REGION Network 19: 9
   RUNG wire#powerrail
      I_Contact( "AlwaysFALSE" )
      Contact( "DB_Data".F9.Sensor_Correct_Position )
      wire#w1
      Contact( "Q_Door_Open" )
      { S7_Templates := "SrcType := Int" } LT_Contact(in1 := "Simu_Door_F9", in2 := 10)
      Contact( "Clock_1Hz" )
      P_Trig( "P108" )
      Add(in1 := "Simu_Door_F9", in2 := 1, out => "Simu_Door_F9")
   END_RUNG
   RUNG wire#w1
      Contact( "Q_Door_Close" )
      { S7_Templates := "SrcType := Int" } GT_Contact(in1 := "Simu_Door_F9", in2 := 0)
      Contact( "Clock_1Hz" )
      P_Trig( "P109" )
      Sub(in1 := "Simu_Door_F9", in2 := 1, out => "Simu_Door_F9")
   END_RUNG
   // the same network as SCL:
   #_w1 := NOT "AlwaysFALSE" AND "DB_Data".F9.Sensor_Correct_Position;
   #_w2 := #_w1 AND "Q_Door_Open" AND ("Simu_Door_F9" < 10) AND "Clock_1Hz";
   #_w3 := #_w2 AND NOT "P108";   // rising edge
   "P108" := #_w2;
   IF #_w3 THEN "Simu_Door_F9" := "Simu_Door_F9" + 1; END_IF;
   #_w4 := #_w1 AND "Q_Door_Close" AND ("Simu_Door_F9" > 0) AND "Clock_1Hz";
   #_w5 := #_w4 AND NOT "P109";   // rising edge
   "P109" := #_w4;
   IF #_w5 THEN "Simu_Door_F9" := "Simu_Door_F9" - 1; END_IF;
END_REGION

REGION Network 20: 9
   RUNG wire#powerrail
      I_Contact( "AlwaysFALSE" )
      Contact( "DB_Data".F9.Position )
      wire#w1
      { S7_Templates := "SrcType := Int" } GE_Contact(in1 := "Simu_Door_F9", in2 := 10)
      Coil( "DB_Data".F9.Door_Opened )
   END_RUNG
   RUNG wire#w1
      { S7_Templates := "SrcType := Int" } LE_Contact(in1 := "Simu_Door_F9", in2 := 0)
      Coil( "DB_Data".F9.Door_Closed )
   END_RUNG
   // the same network as SCL:
   #_w1 := NOT "AlwaysFALSE" AND "DB_Data".F9.Position;
   "DB_Data".F9.Door_Opened := #_w1 AND ("Simu_Door_F9" >= 10);
   "DB_Data".F9.Door_Closed := #_w1 AND ("Simu_Door_F9" <= 0);
END_REGION

REGION Network 21: 10
   RUNG wire#powerrail
      I_Contact( "AlwaysFALSE" )
      Contact( "DB_Data".F10.Sensor_Correct_Position )
      wire#w1
      Contact( "Q_Door_Open" )
      { S7_Templates := "SrcType := Int" } LT_Contact(in1 := "Simu_Door_F10", in2 := 10)
      Contact( "Clock_1Hz" )
      P_Trig( "P110" )
      Add(in1 := "Simu_Door_F10", in2 := 1, out => "Simu_Door_F10")
   END_RUNG
   RUNG wire#w1
      Contact( "Q_Door_Close" )
      { S7_Templates := "SrcType := Int" } GT_Contact(in1 := "Simu_Door_F10", in2 := 0)
      Contact( "Clock_1Hz" )
      P_Trig( "P111" )
      Sub(in1 := "Simu_Door_F10", in2 := 1, out => "Simu_Door_F10")
   END_RUNG
   // the same network as SCL:
   #_w1 := NOT "AlwaysFALSE" AND "DB_Data".F10.Sensor_Correct_Position;
   #_w2 := #_w1 AND "Q_Door_Open" AND ("Simu_Door_F10" < 10) AND "Clock_1Hz";
   #_w3 := #_w2 AND NOT "P110";   // rising edge
   "P110" := #_w2;
   IF #_w3 THEN "Simu_Door_F10" := "Simu_Door_F10" + 1; END_IF;
   #_w4 := #_w1 AND "Q_Door_Close" AND ("Simu_Door_F10" > 0) AND "Clock_1Hz";
   #_w5 := #_w4 AND NOT "P111";   // rising edge
   "P111" := #_w4;
   IF #_w5 THEN "Simu_Door_F10" := "Simu_Door_F10" - 1; END_IF;
END_REGION

REGION Network 22: 10
   RUNG wire#powerrail
      I_Contact( "AlwaysFALSE" )
      Contact( "DB_Data".F10.Position )
      wire#w1
      { S7_Templates := "SrcType := Int" } GE_Contact(in1 := "Simu_Door_F10", in2 := 10)
      Coil( "DB_Data".F10.Door_Opened )
   END_RUNG
   RUNG wire#w1
      { S7_Templates := "SrcType := Int" } LE_Contact(in1 := "Simu_Door_F10", in2 := 0)
      Coil( "DB_Data".F10.Door_Closed )
   END_RUNG
   // the same network as SCL:
   #_w1 := NOT "AlwaysFALSE" AND "DB_Data".F10.Position;
   "DB_Data".F10.Door_Opened := #_w1 AND ("Simu_Door_F10" >= 10);
   "DB_Data".F10.Door_Closed := #_w1 AND ("Simu_Door_F10" <= 0);
END_REGION

REGION Network 23: 11
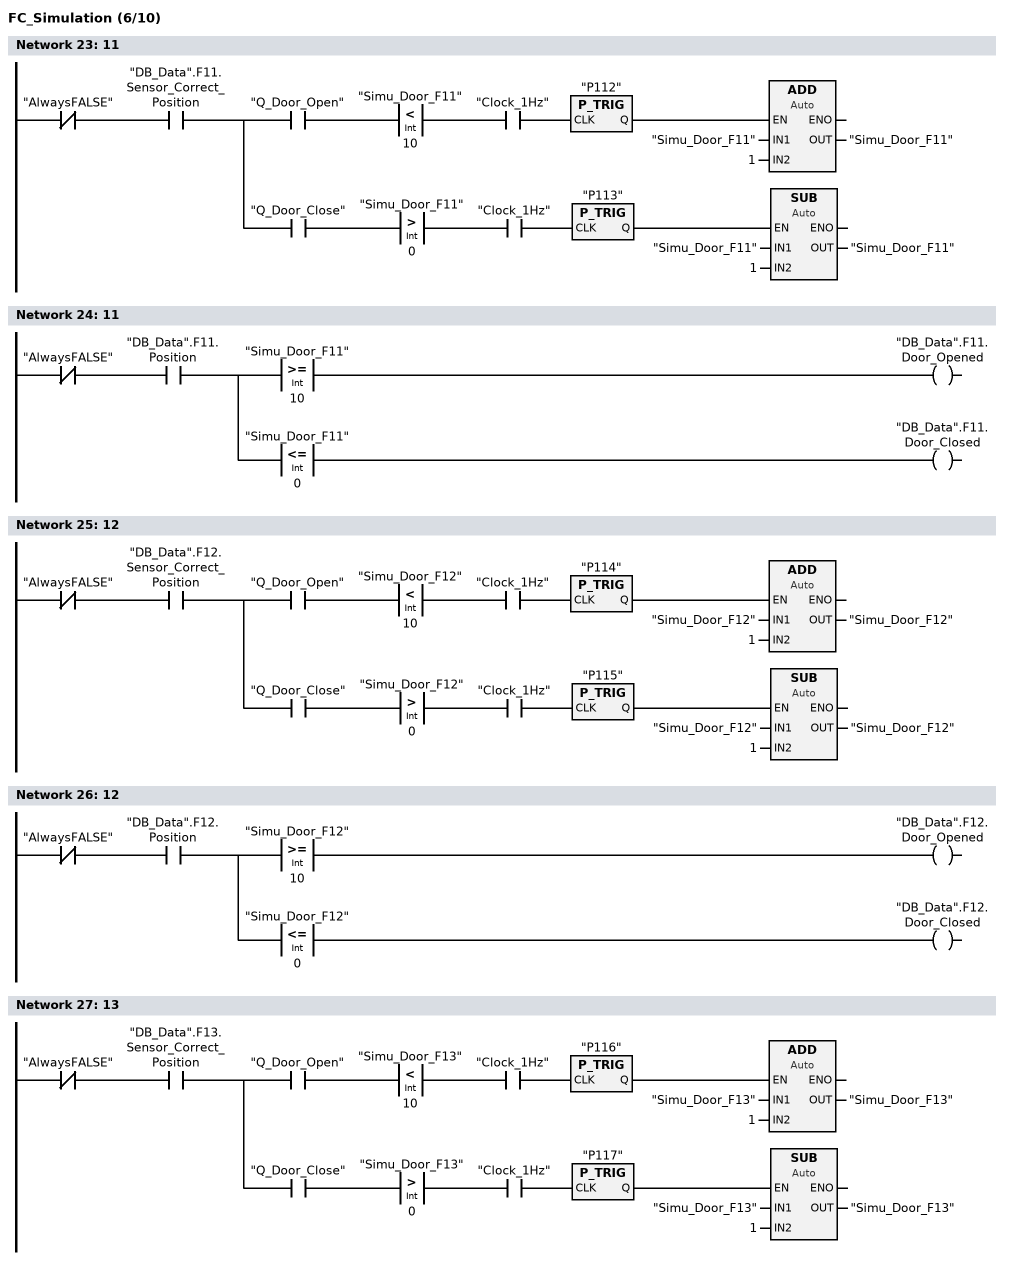
   RUNG wire#powerrail
      I_Contact( "AlwaysFALSE" )
      Contact( "DB_Data".F11.Sensor_Correct_Position )
      wire#w1
      Contact( "Q_Door_Open" )
      { S7_Templates := "SrcType := Int" } LT_Contact(in1 := "Simu_Door_F11", in2 := 10)
      Contact( "Clock_1Hz" )
      P_Trig( "P112" )
      Add(in1 := "Simu_Door_F11", in2 := 1, out => "Simu_Door_F11")
   END_RUNG
   RUNG wire#w1
      Contact( "Q_Door_Close" )
      { S7_Templates := "SrcType := Int" } GT_Contact(in1 := "Simu_Door_F11", in2 := 0)
      Contact( "Clock_1Hz" )
      P_Trig( "P113" )
      Sub(in1 := "Simu_Door_F11", in2 := 1, out => "Simu_Door_F11")
   END_RUNG
   // the same network as SCL:
   #_w1 := NOT "AlwaysFALSE" AND "DB_Data".F11.Sensor_Correct_Position;
   #_w2 := #_w1 AND "Q_Door_Open" AND ("Simu_Door_F11" < 10) AND "Clock_1Hz";
   #_w3 := #_w2 AND NOT "P112";   // rising edge
   "P112" := #_w2;
   IF #_w3 THEN "Simu_Door_F11" := "Simu_Door_F11" + 1; END_IF;
   #_w4 := #_w1 AND "Q_Door_Close" AND ("Simu_Door_F11" > 0) AND "Clock_1Hz";
   #_w5 := #_w4 AND NOT "P113";   // rising edge
   "P113" := #_w4;
   IF #_w5 THEN "Simu_Door_F11" := "Simu_Door_F11" - 1; END_IF;
END_REGION

REGION Network 24: 11
   RUNG wire#powerrail
      I_Contact( "AlwaysFALSE" )
      Contact( "DB_Data".F11.Position )
      wire#w1
      { S7_Templates := "SrcType := Int" } GE_Contact(in1 := "Simu_Door_F11", in2 := 10)
      Coil( "DB_Data".F11.Door_Opened )
   END_RUNG
   RUNG wire#w1
      { S7_Templates := "SrcType := Int" } LE_Contact(in1 := "Simu_Door_F11", in2 := 0)
      Coil( "DB_Data".F11.Door_Closed )
   END_RUNG
   // the same network as SCL:
   #_w1 := NOT "AlwaysFALSE" AND "DB_Data".F11.Position;
   "DB_Data".F11.Door_Opened := #_w1 AND ("Simu_Door_F11" >= 10);
   "DB_Data".F11.Door_Closed := #_w1 AND ("Simu_Door_F11" <= 0);
END_REGION

REGION Network 25: 12
   RUNG wire#powerrail
      I_Contact( "AlwaysFALSE" )
      Contact( "DB_Data".F12.Sensor_Correct_Position )
      wire#w1
      Contact( "Q_Door_Open" )
      { S7_Templates := "SrcType := Int" } LT_Contact(in1 := "Simu_Door_F12", in2 := 10)
      Contact( "Clock_1Hz" )
      P_Trig( "P114" )
      Add(in1 := "Simu_Door_F12", in2 := 1, out => "Simu_Door_F12")
   END_RUNG
   RUNG wire#w1
      Contact( "Q_Door_Close" )
      { S7_Templates := "SrcType := Int" } GT_Contact(in1 := "Simu_Door_F12", in2 := 0)
      Contact( "Clock_1Hz" )
      P_Trig( "P115" )
      Sub(in1 := "Simu_Door_F12", in2 := 1, out => "Simu_Door_F12")
   END_RUNG
   // the same network as SCL:
   #_w1 := NOT "AlwaysFALSE" AND "DB_Data".F12.Sensor_Correct_Position;
   #_w2 := #_w1 AND "Q_Door_Open" AND ("Simu_Door_F12" < 10) AND "Clock_1Hz";
   #_w3 := #_w2 AND NOT "P114";   // rising edge
   "P114" := #_w2;
   IF #_w3 THEN "Simu_Door_F12" := "Simu_Door_F12" + 1; END_IF;
   #_w4 := #_w1 AND "Q_Door_Close" AND ("Simu_Door_F12" > 0) AND "Clock_1Hz";
   #_w5 := #_w4 AND NOT "P115";   // rising edge
   "P115" := #_w4;
   IF #_w5 THEN "Simu_Door_F12" := "Simu_Door_F12" - 1; END_IF;
END_REGION

REGION Network 26: 12
   RUNG wire#powerrail
      I_Contact( "AlwaysFALSE" )
      Contact( "DB_Data".F12.Position )
      wire#w1
      { S7_Templates := "SrcType := Int" } GE_Contact(in1 := "Simu_Door_F12", in2 := 10)
      Coil( "DB_Data".F12.Door_Opened )
   END_RUNG
   RUNG wire#w1
      { S7_Templates := "SrcType := Int" } LE_Contact(in1 := "Simu_Door_F12", in2 := 0)
      Coil( "DB_Data".F12.Door_Closed )
   END_RUNG
   // the same network as SCL:
   #_w1 := NOT "AlwaysFALSE" AND "DB_Data".F12.Position;
   "DB_Data".F12.Door_Opened := #_w1 AND ("Simu_Door_F12" >= 10);
   "DB_Data".F12.Door_Closed := #_w1 AND ("Simu_Door_F12" <= 0);
END_REGION

REGION Network 27: 13
   RUNG wire#powerrail
      I_Contact( "AlwaysFALSE" )
      Contact( "DB_Data".F13.Sensor_Correct_Position )
      wire#w1
      Contact( "Q_Door_Open" )
      { S7_Templates := "SrcType := Int" } LT_Contact(in1 := "Simu_Door_F13", in2 := 10)
      Contact( "Clock_1Hz" )
      P_Trig( "P116" )
      Add(in1 := "Simu_Door_F13", in2 := 1, out => "Simu_Door_F13")
   END_RUNG
   RUNG wire#w1
      Contact( "Q_Door_Close" )
      { S7_Templates := "SrcType := Int" } GT_Contact(in1 := "Simu_Door_F13", in2 := 0)
      Contact( "Clock_1Hz" )
      P_Trig( "P117" )
      Sub(in1 := "Simu_Door_F13", in2 := 1, out => "Simu_Door_F13")
   END_RUNG
   // the same network as SCL:
   #_w1 := NOT "AlwaysFALSE" AND "DB_Data".F13.Sensor_Correct_Position;
   #_w2 := #_w1 AND "Q_Door_Open" AND ("Simu_Door_F13" < 10) AND "Clock_1Hz";
   #_w3 := #_w2 AND NOT "P116";   // rising edge
   "P116" := #_w2;
   IF #_w3 THEN "Simu_Door_F13" := "Simu_Door_F13" + 1; END_IF;
   #_w4 := #_w1 AND "Q_Door_Close" AND ("Simu_Door_F13" > 0) AND "Clock_1Hz";
   #_w5 := #_w4 AND NOT "P117";   // rising edge
   "P117" := #_w4;
   IF #_w5 THEN "Simu_Door_F13" := "Simu_Door_F13" - 1; END_IF;
END_REGION

REGION Network 28: 13
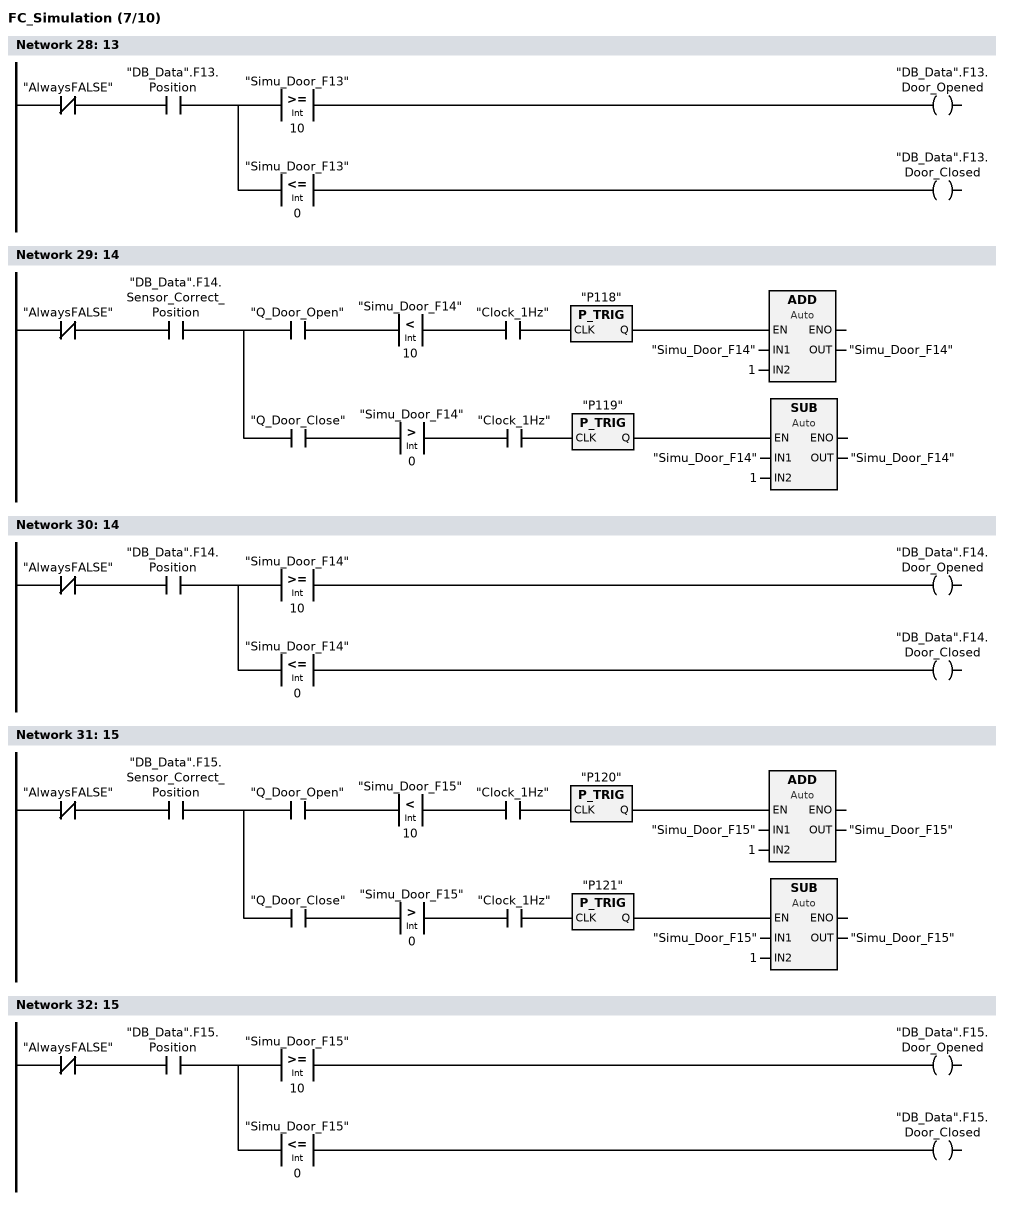
   RUNG wire#powerrail
      I_Contact( "AlwaysFALSE" )
      Contact( "DB_Data".F13.Position )
      wire#w1
      { S7_Templates := "SrcType := Int" } GE_Contact(in1 := "Simu_Door_F13", in2 := 10)
      Coil( "DB_Data".F13.Door_Opened )
   END_RUNG
   RUNG wire#w1
      { S7_Templates := "SrcType := Int" } LE_Contact(in1 := "Simu_Door_F13", in2 := 0)
      Coil( "DB_Data".F13.Door_Closed )
   END_RUNG
   // the same network as SCL:
   #_w1 := NOT "AlwaysFALSE" AND "DB_Data".F13.Position;
   "DB_Data".F13.Door_Opened := #_w1 AND ("Simu_Door_F13" >= 10);
   "DB_Data".F13.Door_Closed := #_w1 AND ("Simu_Door_F13" <= 0);
END_REGION

REGION Network 29: 14
   RUNG wire#powerrail
      I_Contact( "AlwaysFALSE" )
      Contact( "DB_Data".F14.Sensor_Correct_Position )
      wire#w1
      Contact( "Q_Door_Open" )
      { S7_Templates := "SrcType := Int" } LT_Contact(in1 := "Simu_Door_F14", in2 := 10)
      Contact( "Clock_1Hz" )
      P_Trig( "P118" )
      Add(in1 := "Simu_Door_F14", in2 := 1, out => "Simu_Door_F14")
   END_RUNG
   RUNG wire#w1
      Contact( "Q_Door_Close" )
      { S7_Templates := "SrcType := Int" } GT_Contact(in1 := "Simu_Door_F14", in2 := 0)
      Contact( "Clock_1Hz" )
      P_Trig( "P119" )
      Sub(in1 := "Simu_Door_F14", in2 := 1, out => "Simu_Door_F14")
   END_RUNG
   // the same network as SCL:
   #_w1 := NOT "AlwaysFALSE" AND "DB_Data".F14.Sensor_Correct_Position;
   #_w2 := #_w1 AND "Q_Door_Open" AND ("Simu_Door_F14" < 10) AND "Clock_1Hz";
   #_w3 := #_w2 AND NOT "P118";   // rising edge
   "P118" := #_w2;
   IF #_w3 THEN "Simu_Door_F14" := "Simu_Door_F14" + 1; END_IF;
   #_w4 := #_w1 AND "Q_Door_Close" AND ("Simu_Door_F14" > 0) AND "Clock_1Hz";
   #_w5 := #_w4 AND NOT "P119";   // rising edge
   "P119" := #_w4;
   IF #_w5 THEN "Simu_Door_F14" := "Simu_Door_F14" - 1; END_IF;
END_REGION

REGION Network 30: 14
   RUNG wire#powerrail
      I_Contact( "AlwaysFALSE" )
      Contact( "DB_Data".F14.Position )
      wire#w1
      { S7_Templates := "SrcType := Int" } GE_Contact(in1 := "Simu_Door_F14", in2 := 10)
      Coil( "DB_Data".F14.Door_Opened )
   END_RUNG
   RUNG wire#w1
      { S7_Templates := "SrcType := Int" } LE_Contact(in1 := "Simu_Door_F14", in2 := 0)
      Coil( "DB_Data".F14.Door_Closed )
   END_RUNG
   // the same network as SCL:
   #_w1 := NOT "AlwaysFALSE" AND "DB_Data".F14.Position;
   "DB_Data".F14.Door_Opened := #_w1 AND ("Simu_Door_F14" >= 10);
   "DB_Data".F14.Door_Closed := #_w1 AND ("Simu_Door_F14" <= 0);
END_REGION

REGION Network 31: 15
   RUNG wire#powerrail
      I_Contact( "AlwaysFALSE" )
      Contact( "DB_Data".F15.Sensor_Correct_Position )
      wire#w1
      Contact( "Q_Door_Open" )
      { S7_Templates := "SrcType := Int" } LT_Contact(in1 := "Simu_Door_F15", in2 := 10)
      Contact( "Clock_1Hz" )
      P_Trig( "P120" )
      Add(in1 := "Simu_Door_F15", in2 := 1, out => "Simu_Door_F15")
   END_RUNG
   RUNG wire#w1
      Contact( "Q_Door_Close" )
      { S7_Templates := "SrcType := Int" } GT_Contact(in1 := "Simu_Door_F15", in2 := 0)
      Contact( "Clock_1Hz" )
      P_Trig( "P121" )
      Sub(in1 := "Simu_Door_F15", in2 := 1, out => "Simu_Door_F15")
   END_RUNG
   // the same network as SCL:
   #_w1 := NOT "AlwaysFALSE" AND "DB_Data".F15.Sensor_Correct_Position;
   #_w2 := #_w1 AND "Q_Door_Open" AND ("Simu_Door_F15" < 10) AND "Clock_1Hz";
   #_w3 := #_w2 AND NOT "P120";   // rising edge
   "P120" := #_w2;
   IF #_w3 THEN "Simu_Door_F15" := "Simu_Door_F15" + 1; END_IF;
   #_w4 := #_w1 AND "Q_Door_Close" AND ("Simu_Door_F15" > 0) AND "Clock_1Hz";
   #_w5 := #_w4 AND NOT "P121";   // rising edge
   "P121" := #_w4;
   IF #_w5 THEN "Simu_Door_F15" := "Simu_Door_F15" - 1; END_IF;
END_REGION

REGION Network 32: 15
   RUNG wire#powerrail
      I_Contact( "AlwaysFALSE" )
      Contact( "DB_Data".F15.Position )
      wire#w1
      { S7_Templates := "SrcType := Int" } GE_Contact(in1 := "Simu_Door_F15", in2 := 10)
      Coil( "DB_Data".F15.Door_Opened )
   END_RUNG
   RUNG wire#w1
      { S7_Templates := "SrcType := Int" } LE_Contact(in1 := "Simu_Door_F15", in2 := 0)
      Coil( "DB_Data".F15.Door_Closed )
   END_RUNG
   // the same network as SCL:
   #_w1 := NOT "AlwaysFALSE" AND "DB_Data".F15.Position;
   "DB_Data".F15.Door_Opened := #_w1 AND ("Simu_Door_F15" >= 10);
   "DB_Data".F15.Door_Closed := #_w1 AND ("Simu_Door_F15" <= 0);
END_REGION

REGION Network 33: 16
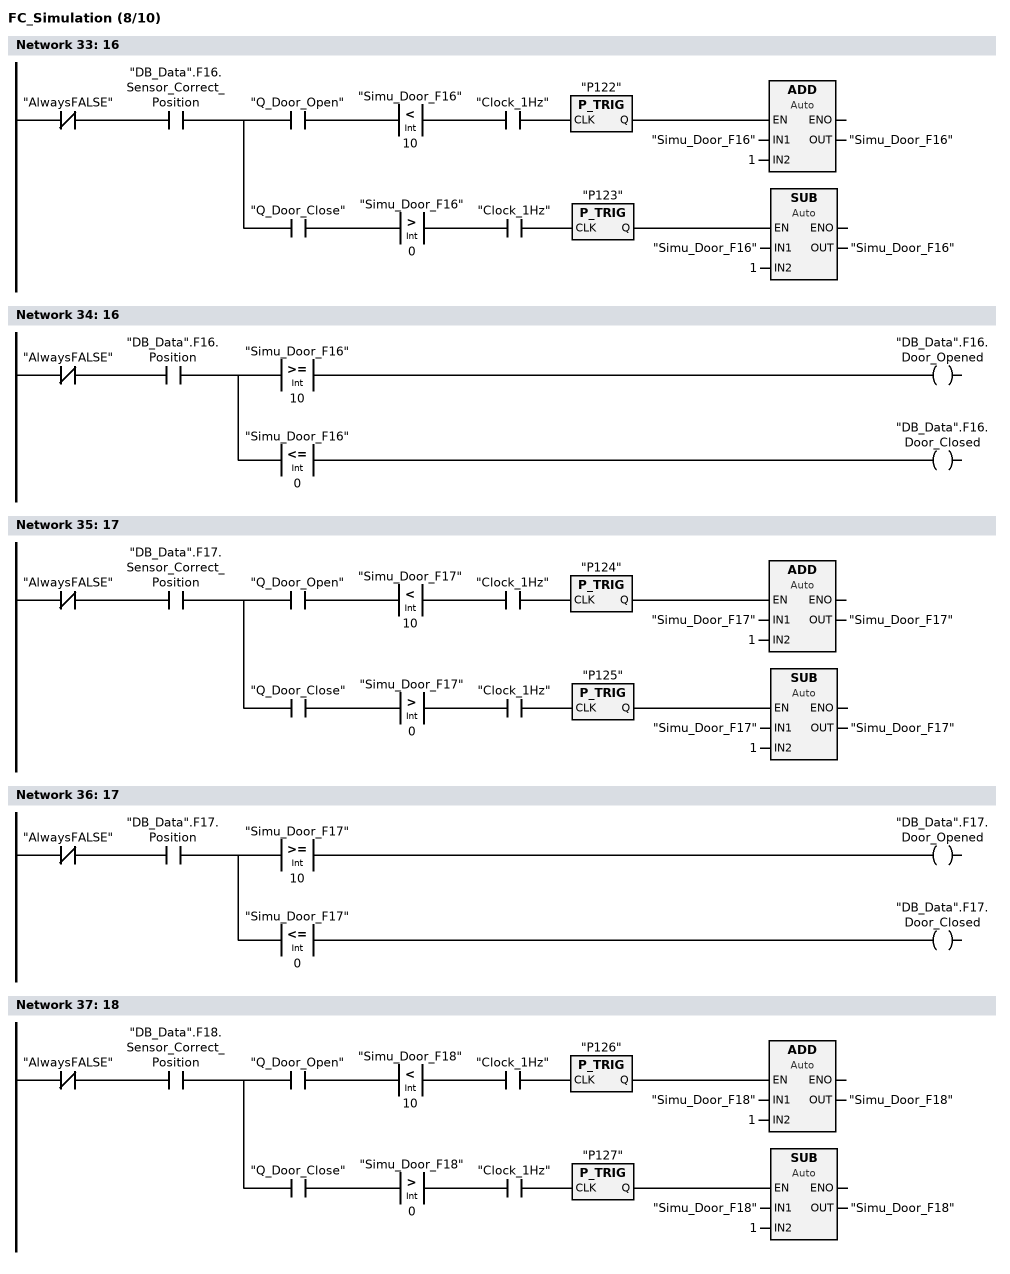
   RUNG wire#powerrail
      I_Contact( "AlwaysFALSE" )
      Contact( "DB_Data".F16.Sensor_Correct_Position )
      wire#w1
      Contact( "Q_Door_Open" )
      { S7_Templates := "SrcType := Int" } LT_Contact(in1 := "Simu_Door_F16", in2 := 10)
      Contact( "Clock_1Hz" )
      P_Trig( "P122" )
      Add(in1 := "Simu_Door_F16", in2 := 1, out => "Simu_Door_F16")
   END_RUNG
   RUNG wire#w1
      Contact( "Q_Door_Close" )
      { S7_Templates := "SrcType := Int" } GT_Contact(in1 := "Simu_Door_F16", in2 := 0)
      Contact( "Clock_1Hz" )
      P_Trig( "P123" )
      Sub(in1 := "Simu_Door_F16", in2 := 1, out => "Simu_Door_F16")
   END_RUNG
   // the same network as SCL:
   #_w1 := NOT "AlwaysFALSE" AND "DB_Data".F16.Sensor_Correct_Position;
   #_w2 := #_w1 AND "Q_Door_Open" AND ("Simu_Door_F16" < 10) AND "Clock_1Hz";
   #_w3 := #_w2 AND NOT "P122";   // rising edge
   "P122" := #_w2;
   IF #_w3 THEN "Simu_Door_F16" := "Simu_Door_F16" + 1; END_IF;
   #_w4 := #_w1 AND "Q_Door_Close" AND ("Simu_Door_F16" > 0) AND "Clock_1Hz";
   #_w5 := #_w4 AND NOT "P123";   // rising edge
   "P123" := #_w4;
   IF #_w5 THEN "Simu_Door_F16" := "Simu_Door_F16" - 1; END_IF;
END_REGION

REGION Network 34: 16
   RUNG wire#powerrail
      I_Contact( "AlwaysFALSE" )
      Contact( "DB_Data".F16.Position )
      wire#w1
      { S7_Templates := "SrcType := Int" } GE_Contact(in1 := "Simu_Door_F16", in2 := 10)
      Coil( "DB_Data".F16.Door_Opened )
   END_RUNG
   RUNG wire#w1
      { S7_Templates := "SrcType := Int" } LE_Contact(in1 := "Simu_Door_F16", in2 := 0)
      Coil( "DB_Data".F16.Door_Closed )
   END_RUNG
   // the same network as SCL:
   #_w1 := NOT "AlwaysFALSE" AND "DB_Data".F16.Position;
   "DB_Data".F16.Door_Opened := #_w1 AND ("Simu_Door_F16" >= 10);
   "DB_Data".F16.Door_Closed := #_w1 AND ("Simu_Door_F16" <= 0);
END_REGION

REGION Network 35: 17
   RUNG wire#powerrail
      I_Contact( "AlwaysFALSE" )
      Contact( "DB_Data".F17.Sensor_Correct_Position )
      wire#w1
      Contact( "Q_Door_Open" )
      { S7_Templates := "SrcType := Int" } LT_Contact(in1 := "Simu_Door_F17", in2 := 10)
      Contact( "Clock_1Hz" )
      P_Trig( "P124" )
      Add(in1 := "Simu_Door_F17", in2 := 1, out => "Simu_Door_F17")
   END_RUNG
   RUNG wire#w1
      Contact( "Q_Door_Close" )
      { S7_Templates := "SrcType := Int" } GT_Contact(in1 := "Simu_Door_F17", in2 := 0)
      Contact( "Clock_1Hz" )
      P_Trig( "P125" )
      Sub(in1 := "Simu_Door_F17", in2 := 1, out => "Simu_Door_F17")
   END_RUNG
   // the same network as SCL:
   #_w1 := NOT "AlwaysFALSE" AND "DB_Data".F17.Sensor_Correct_Position;
   #_w2 := #_w1 AND "Q_Door_Open" AND ("Simu_Door_F17" < 10) AND "Clock_1Hz";
   #_w3 := #_w2 AND NOT "P124";   // rising edge
   "P124" := #_w2;
   IF #_w3 THEN "Simu_Door_F17" := "Simu_Door_F17" + 1; END_IF;
   #_w4 := #_w1 AND "Q_Door_Close" AND ("Simu_Door_F17" > 0) AND "Clock_1Hz";
   #_w5 := #_w4 AND NOT "P125";   // rising edge
   "P125" := #_w4;
   IF #_w5 THEN "Simu_Door_F17" := "Simu_Door_F17" - 1; END_IF;
END_REGION

REGION Network 36: 17
   RUNG wire#powerrail
      I_Contact( "AlwaysFALSE" )
      Contact( "DB_Data".F17.Position )
      wire#w1
      { S7_Templates := "SrcType := Int" } GE_Contact(in1 := "Simu_Door_F17", in2 := 10)
      Coil( "DB_Data".F17.Door_Opened )
   END_RUNG
   RUNG wire#w1
      { S7_Templates := "SrcType := Int" } LE_Contact(in1 := "Simu_Door_F17", in2 := 0)
      Coil( "DB_Data".F17.Door_Closed )
   END_RUNG
   // the same network as SCL:
   #_w1 := NOT "AlwaysFALSE" AND "DB_Data".F17.Position;
   "DB_Data".F17.Door_Opened := #_w1 AND ("Simu_Door_F17" >= 10);
   "DB_Data".F17.Door_Closed := #_w1 AND ("Simu_Door_F17" <= 0);
END_REGION

REGION Network 37: 18
   RUNG wire#powerrail
      I_Contact( "AlwaysFALSE" )
      Contact( "DB_Data".F18.Sensor_Correct_Position )
      wire#w1
      Contact( "Q_Door_Open" )
      { S7_Templates := "SrcType := Int" } LT_Contact(in1 := "Simu_Door_F18", in2 := 10)
      Contact( "Clock_1Hz" )
      P_Trig( "P126" )
      Add(in1 := "Simu_Door_F18", in2 := 1, out => "Simu_Door_F18")
   END_RUNG
   RUNG wire#w1
      Contact( "Q_Door_Close" )
      { S7_Templates := "SrcType := Int" } GT_Contact(in1 := "Simu_Door_F18", in2 := 0)
      Contact( "Clock_1Hz" )
      P_Trig( "P127" )
      Sub(in1 := "Simu_Door_F18", in2 := 1, out => "Simu_Door_F18")
   END_RUNG
   // the same network as SCL:
   #_w1 := NOT "AlwaysFALSE" AND "DB_Data".F18.Sensor_Correct_Position;
   #_w2 := #_w1 AND "Q_Door_Open" AND ("Simu_Door_F18" < 10) AND "Clock_1Hz";
   #_w3 := #_w2 AND NOT "P126";   // rising edge
   "P126" := #_w2;
   IF #_w3 THEN "Simu_Door_F18" := "Simu_Door_F18" + 1; END_IF;
   #_w4 := #_w1 AND "Q_Door_Close" AND ("Simu_Door_F18" > 0) AND "Clock_1Hz";
   #_w5 := #_w4 AND NOT "P127";   // rising edge
   "P127" := #_w4;
   IF #_w5 THEN "Simu_Door_F18" := "Simu_Door_F18" - 1; END_IF;
END_REGION

REGION Network 38: 18
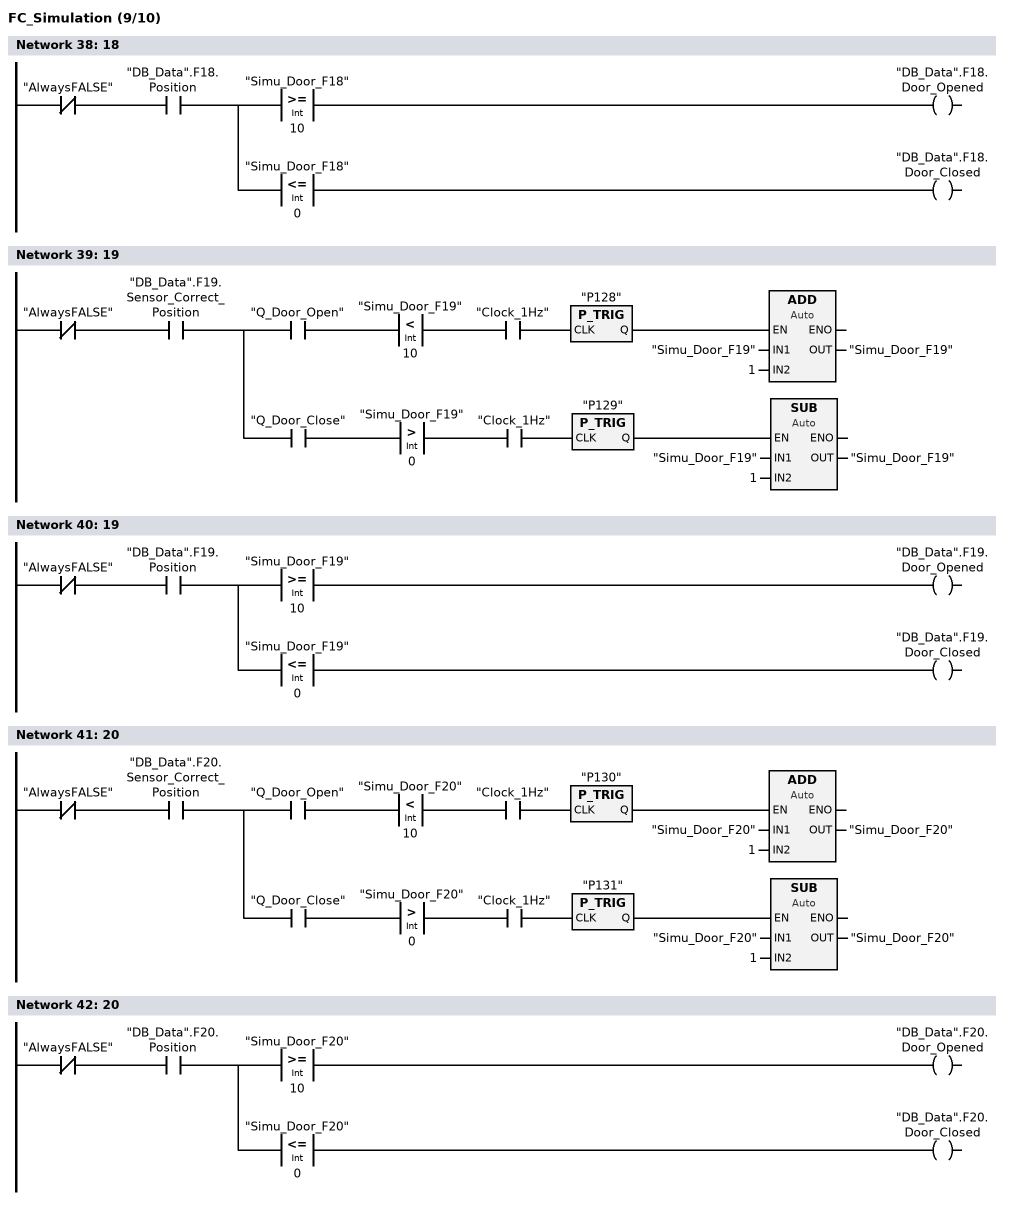
   RUNG wire#powerrail
      I_Contact( "AlwaysFALSE" )
      Contact( "DB_Data".F18.Position )
      wire#w1
      { S7_Templates := "SrcType := Int" } GE_Contact(in1 := "Simu_Door_F18", in2 := 10)
      Coil( "DB_Data".F18.Door_Opened )
   END_RUNG
   RUNG wire#w1
      { S7_Templates := "SrcType := Int" } LE_Contact(in1 := "Simu_Door_F18", in2 := 0)
      Coil( "DB_Data".F18.Door_Closed )
   END_RUNG
   // the same network as SCL:
   #_w1 := NOT "AlwaysFALSE" AND "DB_Data".F18.Position;
   "DB_Data".F18.Door_Opened := #_w1 AND ("Simu_Door_F18" >= 10);
   "DB_Data".F18.Door_Closed := #_w1 AND ("Simu_Door_F18" <= 0);
END_REGION

REGION Network 39: 19
   RUNG wire#powerrail
      I_Contact( "AlwaysFALSE" )
      Contact( "DB_Data".F19.Sensor_Correct_Position )
      wire#w1
      Contact( "Q_Door_Open" )
      { S7_Templates := "SrcType := Int" } LT_Contact(in1 := "Simu_Door_F19", in2 := 10)
      Contact( "Clock_1Hz" )
      P_Trig( "P128" )
      Add(in1 := "Simu_Door_F19", in2 := 1, out => "Simu_Door_F19")
   END_RUNG
   RUNG wire#w1
      Contact( "Q_Door_Close" )
      { S7_Templates := "SrcType := Int" } GT_Contact(in1 := "Simu_Door_F19", in2 := 0)
      Contact( "Clock_1Hz" )
      P_Trig( "P129" )
      Sub(in1 := "Simu_Door_F19", in2 := 1, out => "Simu_Door_F19")
   END_RUNG
   // the same network as SCL:
   #_w1 := NOT "AlwaysFALSE" AND "DB_Data".F19.Sensor_Correct_Position;
   #_w2 := #_w1 AND "Q_Door_Open" AND ("Simu_Door_F19" < 10) AND "Clock_1Hz";
   #_w3 := #_w2 AND NOT "P128";   // rising edge
   "P128" := #_w2;
   IF #_w3 THEN "Simu_Door_F19" := "Simu_Door_F19" + 1; END_IF;
   #_w4 := #_w1 AND "Q_Door_Close" AND ("Simu_Door_F19" > 0) AND "Clock_1Hz";
   #_w5 := #_w4 AND NOT "P129";   // rising edge
   "P129" := #_w4;
   IF #_w5 THEN "Simu_Door_F19" := "Simu_Door_F19" - 1; END_IF;
END_REGION

REGION Network 40: 19
   RUNG wire#powerrail
      I_Contact( "AlwaysFALSE" )
      Contact( "DB_Data".F19.Position )
      wire#w1
      { S7_Templates := "SrcType := Int" } GE_Contact(in1 := "Simu_Door_F19", in2 := 10)
      Coil( "DB_Data".F19.Door_Opened )
   END_RUNG
   RUNG wire#w1
      { S7_Templates := "SrcType := Int" } LE_Contact(in1 := "Simu_Door_F19", in2 := 0)
      Coil( "DB_Data".F19.Door_Closed )
   END_RUNG
   // the same network as SCL:
   #_w1 := NOT "AlwaysFALSE" AND "DB_Data".F19.Position;
   "DB_Data".F19.Door_Opened := #_w1 AND ("Simu_Door_F19" >= 10);
   "DB_Data".F19.Door_Closed := #_w1 AND ("Simu_Door_F19" <= 0);
END_REGION

REGION Network 41: 20
   RUNG wire#powerrail
      I_Contact( "AlwaysFALSE" )
      Contact( "DB_Data".F20.Sensor_Correct_Position )
      wire#w1
      Contact( "Q_Door_Open" )
      { S7_Templates := "SrcType := Int" } LT_Contact(in1 := "Simu_Door_F20", in2 := 10)
      Contact( "Clock_1Hz" )
      P_Trig( "P130" )
      Add(in1 := "Simu_Door_F20", in2 := 1, out => "Simu_Door_F20")
   END_RUNG
   RUNG wire#w1
      Contact( "Q_Door_Close" )
      { S7_Templates := "SrcType := Int" } GT_Contact(in1 := "Simu_Door_F20", in2 := 0)
      Contact( "Clock_1Hz" )
      P_Trig( "P131" )
      Sub(in1 := "Simu_Door_F20", in2 := 1, out => "Simu_Door_F20")
   END_RUNG
   // the same network as SCL:
   #_w1 := NOT "AlwaysFALSE" AND "DB_Data".F20.Sensor_Correct_Position;
   #_w2 := #_w1 AND "Q_Door_Open" AND ("Simu_Door_F20" < 10) AND "Clock_1Hz";
   #_w3 := #_w2 AND NOT "P130";   // rising edge
   "P130" := #_w2;
   IF #_w3 THEN "Simu_Door_F20" := "Simu_Door_F20" + 1; END_IF;
   #_w4 := #_w1 AND "Q_Door_Close" AND ("Simu_Door_F20" > 0) AND "Clock_1Hz";
   #_w5 := #_w4 AND NOT "P131";   // rising edge
   "P131" := #_w4;
   IF #_w5 THEN "Simu_Door_F20" := "Simu_Door_F20" - 1; END_IF;
END_REGION

REGION Network 42: 20
   RUNG wire#powerrail
      I_Contact( "AlwaysFALSE" )
      Contact( "DB_Data".F20.Position )
      wire#w1
      { S7_Templates := "SrcType := Int" } GE_Contact(in1 := "Simu_Door_F20", in2 := 10)
      Coil( "DB_Data".F20.Door_Opened )
   END_RUNG
   RUNG wire#w1
      { S7_Templates := "SrcType := Int" } LE_Contact(in1 := "Simu_Door_F20", in2 := 0)
      Coil( "DB_Data".F20.Door_Closed )
   END_RUNG
   // the same network as SCL:
   #_w1 := NOT "AlwaysFALSE" AND "DB_Data".F20.Position;
   "DB_Data".F20.Door_Opened := #_w1 AND ("Simu_Door_F20" >= 10);
   "DB_Data".F20.Door_Closed := #_w1 AND ("Simu_Door_F20" <= 0);
END_REGION

REGION Network 43: Mô phỏng LS cửa buồng thang
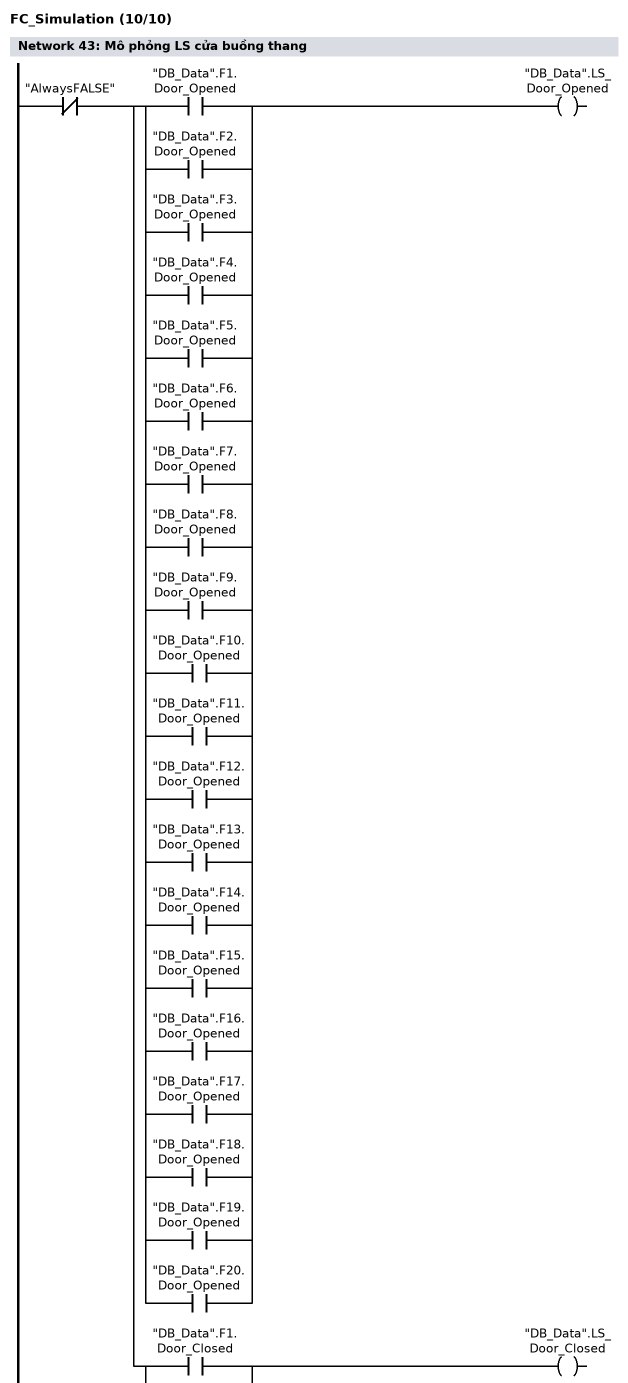
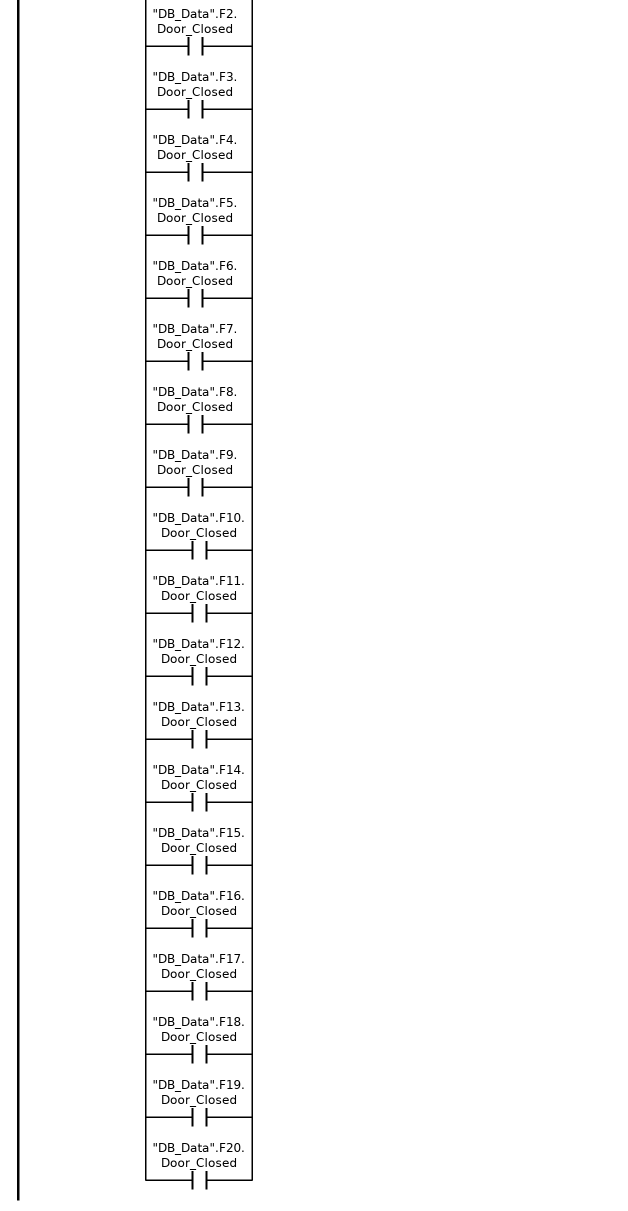
   RUNG wire#powerrail
      I_Contact( "AlwaysFALSE" )
      wire#w1
      Contact( "DB_Data".F1.Door_Opened )
      wire#w2
      Coil( "DB_Data".LS_Door_Opened )
   END_RUNG
   RUNG wire#w1
      Contact( "DB_Data".F2.Door_Opened )
   END_RUNG wire#w2
   RUNG wire#w1
      Contact( "DB_Data".F3.Door_Opened )
   END_RUNG wire#w2
   RUNG wire#w1
      Contact( "DB_Data".F4.Door_Opened )
   END_RUNG wire#w2
   RUNG wire#w1
      Contact( "DB_Data".F5.Door_Opened )
   END_RUNG wire#w2
   RUNG wire#w1
      Contact( "DB_Data".F6.Door_Opened )
   END_RUNG wire#w2
   RUNG wire#w1
      Contact( "DB_Data".F7.Door_Opened )
   END_RUNG wire#w2
   RUNG wire#w1
      Contact( "DB_Data".F8.Door_Opened )
   END_RUNG wire#w2
   RUNG wire#w1
      Contact( "DB_Data".F9.Door_Opened )
   END_RUNG wire#w2
   RUNG wire#w1
      Contact( "DB_Data".F10.Door_Opened )
   END_RUNG wire#w2
   RUNG wire#w1
      Contact( "DB_Data".F11.Door_Opened )
   END_RUNG wire#w2
   RUNG wire#w1
      Contact( "DB_Data".F12.Door_Opened )
   END_RUNG wire#w2
   RUNG wire#w1
      Contact( "DB_Data".F13.Door_Opened )
   END_RUNG wire#w2
   RUNG wire#w1
      Contact( "DB_Data".F14.Door_Opened )
   END_RUNG wire#w2
   RUNG wire#w1
      Contact( "DB_Data".F15.Door_Opened )
   END_RUNG wire#w2
   RUNG wire#w1
      Contact( "DB_Data".F16.Door_Opened )
   END_RUNG wire#w2
   RUNG wire#w1
      Contact( "DB_Data".F17.Door_Opened )
   END_RUNG wire#w2
   RUNG wire#w1
      Contact( "DB_Data".F18.Door_Opened )
   END_RUNG wire#w2
   RUNG wire#w1
      Contact( "DB_Data".F19.Door_Opened )
   END_RUNG wire#w2
   RUNG wire#w1
      Contact( "DB_Data".F20.Door_Opened )
   END_RUNG wire#w2
   RUNG wire#w1
      Contact( "DB_Data".F1.Door_Closed )
      wire#w3
      Coil( "DB_Data".LS_Door_Closed )
   END_RUNG
   RUNG wire#w1
      Contact( "DB_Data".F2.Door_Closed )
   END_RUNG wire#w3
   RUNG wire#w1
      Contact( "DB_Data".F3.Door_Closed )
   END_RUNG wire#w3
   RUNG wire#w1
      Contact( "DB_Data".F4.Door_Closed )
   END_RUNG wire#w3
   RUNG wire#w1
      Contact( "DB_Data".F5.Door_Closed )
   END_RUNG wire#w3
   RUNG wire#w1
      Contact( "DB_Data".F6.Door_Closed )
   END_RUNG wire#w3
   RUNG wire#w1
      Contact( "DB_Data".F7.Door_Closed )
   END_RUNG wire#w3
   RUNG wire#w1
      Contact( "DB_Data".F8.Door_Closed )
   END_RUNG wire#w3
   RUNG wire#w1
      Contact( "DB_Data".F9.Door_Closed )
   END_RUNG wire#w3
   RUNG wire#w1
      Contact( "DB_Data".F10.Door_Closed )
   END_RUNG wire#w3
   RUNG wire#w1
      Contact( "DB_Data".F11.Door_Closed )
   END_RUNG wire#w3
   RUNG wire#w1
      Contact( "DB_Data".F12.Door_Closed )
   END_RUNG wire#w3
   RUNG wire#w1
      Contact( "DB_Data".F13.Door_Closed )
   END_RUNG wire#w3
   RUNG wire#w1
      Contact( "DB_Data".F14.Door_Closed )
   END_RUNG wire#w3
   RUNG wire#w1
      Contact( "DB_Data".F15.Door_Closed )
   END_RUNG wire#w3
   RUNG wire#w1
      Contact( "DB_Data".F16.Door_Closed )
   END_RUNG wire#w3
   RUNG wire#w1
      Contact( "DB_Data".F17.Door_Closed )
   END_RUNG wire#w3
   RUNG wire#w1
      Contact( "DB_Data".F18.Door_Closed )
   END_RUNG wire#w3
   RUNG wire#w1
      Contact( "DB_Data".F19.Door_Closed )
   END_RUNG wire#w3
   RUNG wire#w1
      Contact( "DB_Data".F20.Door_Closed )
   END_RUNG wire#w3
   // the same network as SCL:
   "DB_Data".LS_Door_Opened := NOT "AlwaysFALSE" AND ("DB_Data".F1.Door_Opened OR "DB_Data".F2.Door_Opened OR "DB_Data".F3.Door_Opened OR "DB_Data".F4.Door_Opened OR "DB_Data".F5.Door_Opened OR "DB_Data".F6.Door_Opened OR "DB_Data".F7.Door_Opened OR "DB_Data".F8.Door_Opened OR "DB_Data".F9.Door_Opened OR "DB_Data".F10.Door_Opened OR "DB_Data".F11.Door_Opened OR "DB_Data".F12.Door_Opened OR "DB_Data".F13.Door_Opened OR "DB_Data".F14.Door_Opened OR "DB_Data".F15.Door_Opened OR "DB_Data".F16.Door_Opened OR "DB_Data".F17.Door_Opened OR "DB_Data".F18.Door_Opened OR "DB_Data".F19.Door_Opened OR "DB_Data".F20.Door_Opened);
   "DB_Data".LS_Door_Closed := NOT "AlwaysFALSE" AND ("DB_Data".F1.Door_Closed OR "DB_Data".F2.Door_Closed OR "DB_Data".F3.Door_Closed OR "DB_Data".F4.Door_Closed OR "DB_Data".F5.Door_Closed OR "DB_Data".F6.Door_Closed OR "DB_Data".F7.Door_Closed OR "DB_Data".F8.Door_Closed OR "DB_Data".F9.Door_Closed OR "DB_Data".F10.Door_Closed OR "DB_Data".F11.Door_Closed OR "DB_Data".F12.Door_Closed OR "DB_Data".F13.Door_Closed OR "DB_Data".F14.Door_Closed OR "DB_Data".F15.Door_Closed OR "DB_Data".F16.Door_Closed OR "DB_Data".F17.Door_Closed OR "DB_Data".F18.Door_Closed OR "DB_Data".F19.Door_Closed OR "DB_Data".F20.Door_Closed);
END_REGION
END_FUNCTION

ORGANIZATION_BLOCK "Main"   // OB1, LAD, ProgramCycle
TITLE = "Main Program Sweep (Cycle)"
{ S7_Optimized_Access := 'TRUE' }
VERSION : 0.1
   VAR_INPUT
      Initial_Call : Bool;   // Initial call of this OB
      Remanence : Bool;   // =True, if remanent data are available
   END_VAR
BEGIN

REGION Network 1: Gọi chương trình con nút nhấn
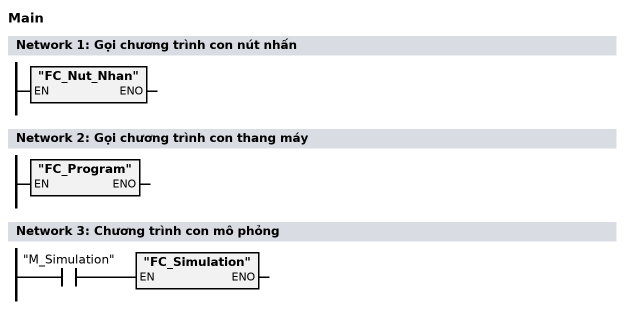
   RUNG wire#powerrail
      "FC_Nut_Nhan"()
   END_RUNG
   // the same network as SCL:
   "FC_Nut_Nhan"();
END_REGION

REGION Network 2: Gọi chương trình con thang máy
   RUNG wire#powerrail
      "FC_Program"()
   END_RUNG
   // the same network as SCL:
   "FC_Program"();
END_REGION

REGION Network 3: Chương trình con mô phỏng
   RUNG wire#powerrail
      Contact( "M_Simulation" )
      "FC_Simulation"()
   END_RUNG
   // the same network as SCL:
   IF "M_Simulation" THEN "FC_Simulation"(); END_IF;
END_REGION
END_ORGANIZATION_BLOCK

(* ===== HMI "HMI_RT_1" =====
system functions are stored by id; their names below are inferred from use
connection "HMI_Connection_1": ETHERNET, S7_1200_OMS

HMI tags "Default tag table"
   "M_Simulation" : Bool = PLC M_Simulation AT %M10.0, 1 s
   "Simu_Eleveytor" : Int = PLC Simu_Eleveytor AT %MW100, 1 s
   "Simu_Door_F1" : Int = PLC Simu_Door_F1 AT %MW102, 1 s
   "Simu_Door_F2" : Int = PLC Simu_Door_F2 AT %MW104, 1 s
   "Simu_Door_F3" : Int = PLC Simu_Door_F3 AT %MW106, 1 s
   "Simu_Door_F4" : Int = PLC Simu_Door_F4 AT %MW108, 1 s
   "DB_Data_F1_I_Button_Up" : Bool = PLC DB_Data.F1.I_Button_Up, 1 s
   "DB_Data_F2_I_Button_Up" : Bool = PLC DB_Data.F2.I_Button_Up, 1 s
   "DB_Data_F2_I_Button_Down" : Bool = PLC DB_Data.F2.I_Button_Down, 1 s
   "DB_Data_F3_I_Button_Up" : Bool = PLC DB_Data.F3.I_Button_Up, 1 s
   "DB_Data_F3_I_Button_Down" : Bool = PLC DB_Data.F3.I_Button_Down, 1 s
   "DB_Data_F4_I_Button_Down" : Bool = PLC DB_Data.F4.I_Button_Down, 1 s
   "DB_Data_Button_Inside_F1" : Bool = PLC DB_Data.Button_Inside_F1, 1 s
   "DB_Data_Button_Inside_F2" : Bool = PLC DB_Data.Button_Inside_F2, 1 s
   "DB_Data_Button_Inside_F3" : Bool = PLC DB_Data.Button_Inside_F3, 1 s
   "DB_Data_Button_Inside_F4" : Bool = PLC DB_Data.Button_Inside_F4, 1 s
   "DB_Data_Button_Inside_Open" : Bool = PLC DB_Data.Button_Inside_Open, 1 s
   "DB_Data_Button_Inside_Close" : Bool = PLC DB_Data.Button_Inside_Close, 1 s
   "DB_Data_F1_Btt_Up_Selected" : Bool = PLC DB_Data.F1.Btt_Up_Selected, 1 s
   "DB_Data_F2_Btt_Up_Selected" : Bool = PLC DB_Data.F2.Btt_Up_Selected, 1 s
   "DB_Data_F2_Btt_Down_Selected" : Bool = PLC DB_Data.F2.Btt_Down_Selected, 1 s
   "DB_Data_F4_Btt_Up_Selected" : Bool = PLC DB_Data.F4.Btt_Up_Selected, 1 s
   "DB_Data_F4_Btt_Down_Selected" : Bool = PLC DB_Data.F4.Btt_Down_Selected, 1 s
   "DB_Data_F3_Btt_Up_Selected" : Bool = PLC DB_Data.F3.Btt_Up_Selected, 1 s
   "DB_Data_F3_Btt_Down_Selected" : Bool = PLC DB_Data.F3.Btt_Down_Selected, 1 s
   "Q_Door_Open" : Bool = PLC Q_Door_Open AT %Q0.0, 1 s
   "Q_Door_Close" : Bool = PLC Q_Door_Close AT %Q0.1, 1 s
   "DB_Data_F1_Sensor_Correct_Position" : Bool = PLC DB_Data.F1.Sensor_Correct_Position, 1 s
   "DB_Data_F2_Sensor_Correct_Position" : Bool = PLC DB_Data.F2.Sensor_Correct_Position, 1 s
   "DB_Data_F3_Sensor_Correct_Position" : Bool = PLC DB_Data.F3.Sensor_Correct_Position, 1 s
   "DB_Data_F4_Sensor_Correct_Position" : Bool = PLC DB_Data.F4.Sensor_Correct_Position, 1 s
   "Display_Inside_F2" : Bool = PLC Display_Inside_F2 AT %M10.1, 1 s
   "Display_Inside_F3" : Bool = PLC Display_Inside_F3 AT %M10.2, 1 s
   "DB_Data_Button_Inside_F5" : Bool = PLC DB_Data.Button_Inside_F5, 1 s
   "DB_Data_Button_Inside_F6" : Bool = PLC DB_Data.Button_Inside_F6, 1 s
   "DB_Data_Button_Inside_F20" : Bool = PLC DB_Data.Button_Inside_F20, 1 s
   "DB_Data_F4_I_Button_Up" : Bool = PLC DB_Data.F4.I_Button_Up, 1 s
   "DB_Data_F5_I_Button_Up" : Bool = PLC DB_Data.F5.I_Button_Up, 1 s
   "DB_Data_F5_I_Button_Down" : Bool = PLC DB_Data.F5.I_Button_Down, 1 s
   "DB_Data_F5_Sensor_Correct_Position" : Bool = PLC DB_Data.F5.Sensor_Correct_Position, 1 s
   "Simu_Door_F5" : Int = PLC Simu_Door_F5 AT %MW110, 1 s
   "DB_Data_F5_Btt_Up_Selected" : Bool = PLC DB_Data.F5.Btt_Up_Selected, 1 s
   "DB_Data_F5_Btt_Down_Selected" : Bool = PLC DB_Data.F5.Btt_Down_Selected, 1 s
   "Display_Inside_F4" : Bool = PLC Display_Inside_F4 AT %M10.3, 1 s
   "Display_Inside_F5" : Bool = PLC Display_Inside_F5 AT %M10.4, 1 s
   "DB_Data_F6_Sensor_Correct_Position" : Bool = PLC DB_Data.F6.Sensor_Correct_Position, 1 s
   "Simu_Door_F6" : Int = PLC Simu_Door_F6 AT %MW112, 1 s
   "DB_Data_F6_Btt_Down_Selected" : Bool = PLC DB_Data.F6.Btt_Down_Selected, 1 s
   "DB_Data_F6_I_Button_Down" : Bool = PLC DB_Data.F6.I_Button_Down, 1 s
   "DB_Data_F6_Btt_Up_Selected" : Bool = PLC DB_Data.F6.Btt_Up_Selected, 1 s
   "DB_Data_F6_I_Button_Up" : Bool = PLC DB_Data.F6.I_Button_Up, 1 s
   "Display_Inside_F6" : Bool = PLC Display_Inside_F6 AT %M10.5, 1 s
   "DB_Data_F7_Sensor_Correct_Position" : Bool = PLC DB_Data.F7.Sensor_Correct_Position, 1 s
   "Simu_Door_F7" : Int = PLC Simu_Door_F7 AT %MW114, 1 s
   "DB_Data_F7_Btt_Up_Selected" : Bool = PLC DB_Data.F7.Btt_Up_Selected, 1 s
   "DB_Data_F7_I_Button_Up" : Bool = PLC DB_Data.F7.I_Button_Up, 1 s
   "DB_Data_F8_I_Button_Up" : Bool = PLC DB_Data.F8.I_Button_Up, 1 s
   "DB_Data_F8_Btt_Up_Selected" : Bool = PLC DB_Data.F8.Btt_Up_Selected, 1 s
   "DB_Data_F7_Btt_Down_Selected" : Bool = PLC DB_Data.F7.Btt_Down_Selected, 1 s
   "DB_Data_F7_I_Button_Down" : Bool = PLC DB_Data.F7.I_Button_Down, 1 s
   "DB_Data_F8_Sensor_Correct_Position" : Bool = PLC DB_Data.F8.Sensor_Correct_Position, 1 s
   "Simu_Door_F8" : Int = PLC Simu_Door_F8 AT %MW116, 1 s
   "DB_Data_F8_Btt_Down_Selected" : Bool = PLC DB_Data.F8.Btt_Down_Selected, 1 s
   "DB_Data_F8_I_Button_Down" : Bool = PLC DB_Data.F8.I_Button_Down, 1 s
   "DB_Data_F9_Sensor_Correct_Position" : Bool = PLC DB_Data.F9.Sensor_Correct_Position, 1 s
   "Simu_Door_F9" : Int = PLC Simu_Door_F9 AT %MW118, 1 s
   "DB_Data_F9_Btt_Up_Selected" : Bool = PLC DB_Data.F9.Btt_Up_Selected, 1 s
   "DB_Data_F9_I_Button_Up" : Bool = PLC DB_Data.F9.I_Button_Up, 1 s
   "DB_Data_F9_I_Button_Down" : Bool = PLC DB_Data.F9.I_Button_Down, 1 s
   "DB_Data_F10_Sensor_Correct_Position" : Bool = PLC DB_Data.F10.Sensor_Correct_Position, 1 s
   "Simu_Door_F10" : Int = PLC Simu_Door_F10 AT %MW120, 1 s
   "DB_Data_F10_Btt_Up_Selected" : Bool = PLC DB_Data.F10.Btt_Up_Selected, 1 s
   "DB_Data_F10_I_Button_Up" : Bool = PLC DB_Data.F10.I_Button_Up, 1 s
   "DB_Data_F10_I_Button_Down" : Bool = PLC DB_Data.F10.I_Button_Down, 1 s
   "DB_Data_F11_Sensor_Correct_Position" : Bool = PLC DB_Data.F11.Sensor_Correct_Position, 1 s
   "Simu_Door_F11" : Int = PLC Simu_Door_F11 AT %MW122, 1 s
   "DB_Data_F11_Btt_Up_Selected" : Bool = PLC DB_Data.F11.Btt_Up_Selected, 1 s
   "DB_Data_F11_I_Button_Up" : Bool = PLC DB_Data.F11.I_Button_Up, 1 s
   "DB_Data_F11_Btt_Down_Selected" : Bool = PLC DB_Data.F11.Btt_Down_Selected, 1 s
   "DB_Data_F11_I_Button_Down" : Bool = PLC DB_Data.F11.I_Button_Down, 1 s
   "DB_Data_F12_Sensor_Correct_Position" : Bool = PLC DB_Data.F12.Sensor_Correct_Position, 1 s
   "Simu_Door_F12" : Int = PLC Simu_Door_F12 AT %MW124, 1 s
   "DB_Data_F12_Btt_Up_Selected" : Bool = PLC DB_Data.F12.Btt_Up_Selected, 1 s
   "DB_Data_F12_I_Button_Up" : Bool = PLC DB_Data.F12.I_Button_Up, 1 s
   "DB_Data_F12_I_Button_Down" : Bool = PLC DB_Data.F12.I_Button_Down, 1 s
   "DB_Data_F12_Btt_Down_Selected" : Bool = PLC DB_Data.F12.Btt_Down_Selected, 1 s
   "Simu_Door_F13" : Int = PLC Simu_Door_F13 AT %MW126, 1 s
   "DB_Data_F13_Sensor_Correct_Position" : Bool = PLC DB_Data.F13.Sensor_Correct_Position, 1 s
   "DB_Data_F13_Btt_Up_Selected" : Bool = PLC DB_Data.F13.Btt_Up_Selected, 1 s
   "DB_Data_F13_I_Button_Up" : Bool = PLC DB_Data.F13.I_Button_Up, 1 s
   "DB_Data_F13_I_Button_Down" : Bool = PLC DB_Data.F13.I_Button_Down, 1 s
   "DB_Data_Button_Inside_F7" : Bool = PLC DB_Data.Button_Inside_F7, 1 s
   "Display_Inside_F7" : Bool = PLC Display_Inside_F7 AT %M10.6, 1 s
   "DB_Data_F10_Btt_Down_Selected" : Bool = PLC DB_Data.F10.Btt_Down_Selected, 1 s
   "DB_Data_F13_Btt_Down_Selected" : Bool = PLC DB_Data.F13.Btt_Down_Selected, 1 s
   "DB_Data_F14_Sensor_Correct_Position" : Bool = PLC DB_Data.F14.Sensor_Correct_Position, 1 s
   "Simu_Door_F14" : Int = PLC Simu_Door_F14 AT %MW128, 1 s
   "DB_Data_F14_Btt_Up_Selected" : Bool = PLC DB_Data.F14.Btt_Up_Selected, 1 s
   "DB_Data_F14_I_Button_Up" : Bool = PLC DB_Data.F14.I_Button_Up, 1 s
   "DB_Data_F14_I_Button_Down" : Bool = PLC DB_Data.F14.I_Button_Down, 1 s
   "DB_Data_F14_Btt_Down_Selected" : Bool = PLC DB_Data.F14.Btt_Down_Selected, 1 s
   "DB_Data_F15_Sensor_Correct_Position" : Bool = PLC DB_Data.F15.Sensor_Correct_Position, 1 s
   "Simu_Door_F15" : Int = PLC Simu_Door_F15 AT %MW130, 1 s
   "DB_Data_F15_Btt_Up_Selected" : Bool = PLC DB_Data.F15.Btt_Up_Selected, 1 s
   "DB_Data_F15_I_Button_Up" : Bool = PLC DB_Data.F15.I_Button_Up, 1 s
   "DB_Data_F15_I_Button_Down" : Bool = PLC DB_Data.F15.I_Button_Down, 1 s
   "DB_Data_F15_Btt_Down_Selected" : Bool = PLC DB_Data.F15.Btt_Down_Selected, 1 s
   "DB_Data_F16_Sensor_Correct_Position" : Bool = PLC DB_Data.F16.Sensor_Correct_Position, 1 s
   "Simu_Door_F16" : Int = PLC Simu_Door_F16 AT %MW132, 1 s
   "DB_Data_F16_Btt_Up_Selected" : Bool = PLC DB_Data.F16.Btt_Up_Selected, 1 s
   "DB_Data_F16_I_Button_Up" : Bool = PLC DB_Data.F16.I_Button_Up, 1 s
   "DB_Data_F16_I_Button_Down" : Bool = PLC DB_Data.F16.I_Button_Down, 1 s
   "DB_Data_F16_Btt_Down_Selected" : Bool = PLC DB_Data.F16.Btt_Down_Selected, 1 s
   "DB_Data_F17_Sensor_Correct_Position" : Bool = PLC DB_Data.F17.Sensor_Correct_Position, 1 s
   "Simu_Door_F17" : Int = PLC Simu_Door_F17 AT %MW134, 1 s
   "DB_Data_F17_Btt_Up_Selected" : Bool = PLC DB_Data.F17.Btt_Up_Selected, 1 s
   "DB_Data_F17_I_Button_Up" : Bool = PLC DB_Data.F17.I_Button_Up, 1 s
   "DB_Data_F17_I_Button_Down" : Bool = PLC DB_Data.F17.I_Button_Down, 1 s
   "DB_Data_F17_Btt_Down_Selected" : Bool = PLC DB_Data.F17.Btt_Down_Selected, 1 s
   "DB_Data_F18_Sensor_Correct_Position" : Bool = PLC DB_Data.F18.Sensor_Correct_Position, 1 s
   "Simu_Door_F18" : Int = PLC Simu_Door_F18 AT %MW136, 1 s
   "DB_Data_F18_Btt_Up_Selected" : Bool = PLC DB_Data.F18.Btt_Up_Selected, 1 s
   "DB_Data_F18_I_Button_Up" : Bool = PLC DB_Data.F18.I_Button_Up, 1 s
   "DB_Data_F18_Btt_Down_Selected" : Bool = PLC DB_Data.F18.Btt_Down_Selected, 1 s
   "DB_Data_F18_I_Button_Down" : Bool = PLC DB_Data.F18.I_Button_Down, 1 s
   "DB_Data_F19_I_Button_Up" : Bool = PLC DB_Data.F19.I_Button_Up, 1 s
   "DB_Data_F19_Btt_Up_Selected" : Bool = PLC DB_Data.F19.Btt_Up_Selected, 1 s
   "DB_Data_F19_Btt_Down_Selected" : Bool = PLC DB_Data.F19.Btt_Down_Selected, 1 s
   "DB_Data_F19_I_Button_Down" : Bool = PLC DB_Data.F19.I_Button_Down, 1 s
   "Simu_Door_F19" : Int = PLC Simu_Door_F19 AT %MW138, 1 s
   "DB_Data_F19_Sensor_Correct_Position" : Bool = PLC DB_Data.F19.Sensor_Correct_Position, 1 s
   "DB_Data_F20_Sensor_Correct_Position" : Bool = PLC DB_Data.F20.Sensor_Correct_Position, 1 s
   "Simu_Door_F20" : Int = PLC Simu_Door_F20 AT %MW140, 1 s
   "DB_Data_F20_Btt_Up_Selected" : Bool = PLC DB_Data.F20.Btt_Up_Selected, 1 s
   "DB_Data_F20_I_Button_Up" : Bool = PLC DB_Data.F20.I_Button_Up, 1 s
   "DB_Data_F20_I_Button_Down" : Bool = PLC DB_Data.F20.I_Button_Down, 1 s
   "DB_Data_F20_Btt_Down_Selected" : Bool = PLC DB_Data.F20.Btt_Down_Selected, 1 s
   "DB_Data_Button_Inside_F8" : Bool = PLC DB_Data.Button_Inside_F8, 1 s
   "Display_Inside_F8" : Bool = PLC Display_Inside_F8 AT %M10.7, 1 s
   "Display_Inside_F9" : Bool = PLC Display_Inside_F9 AT %M11.0, 1 s
   "DB_Data_Button_Inside_F9" : Bool = PLC DB_Data.Button_Inside_F9, 1 s
   "DB_Data_Button_Inside_F10" : Bool = PLC DB_Data.Button_Inside_F10, 1 s
   "Display_Inside_F10" : Bool = PLC Display_Inside_F10 AT %M11.1, 1 s
   "Display_Inside_F11" : Bool = PLC Display_Inside_F11 AT %M11.2, 1 s
   "DB_Data_Button_Inside_F11" : Bool = PLC DB_Data.Button_Inside_F11, 1 s
   "DB_Data_Button_Inside_F12" : Bool = PLC DB_Data.Button_Inside_F12, 1 s
   "Display_Inside_F12" : Bool = PLC Display_Inside_F12 AT %M11.3, 1 s
   "Display_Inside_F13" : Bool = PLC Display_Inside_F13 AT %M11.4, 1 s
   "DB_Data_Button_Inside_F13" : Bool = PLC DB_Data.Button_Inside_F13, 1 s
   "DB_Data_Button_Inside_F14" : Bool = PLC DB_Data.Button_Inside_F14, 1 s
   "Display_Inside_F14" : Bool = PLC Display_Inside_F14 AT %M11.5, 1 s
   "Display_Inside_F15" : Bool = PLC Display_Inside_F15 AT %M11.6, 1 s
   "DB_Data_Button_Inside_F15" : Bool = PLC DB_Data.Button_Inside_F15, 1 s
   "DB_Data_Button_Inside_F16" : Bool = PLC DB_Data.Button_Inside_F16, 1 s
   "Display_Inside_F16" : Bool = PLC Display_Inside_F16 AT %M11.7, 1 s
   "Display_Inside_F17" : Bool = PLC Display_Inside_F17 AT %M12.0, 1 s
   "DB_Data_Button_Inside_F17" : Bool = PLC DB_Data.Button_Inside_F17, 1 s
   "DB_Data_Button_Inside_F18" : Bool = PLC DB_Data.Button_Inside_F18, 1 s
   "Display_Inside_F18" : Bool = PLC Display_Inside_F18 AT %M12.1, 1 s
   "DB_Data_Button_Inside_F19" : Bool = PLC DB_Data.Button_Inside_F19, 1 s
   "Display_Inside_F19" : Bool = PLC Display_Inside_F19 AT %M12.2, 1 s

screen "Screen_1" 1024x1279
   Button "Button_7" at 272,845 size 25x24; TextOff 'v'
      on Press: SetBit("DB_Data_F4_I_Button_Down")
      on Release: ResetBit("DB_Data_F4_I_Button_Down")
      Appearance <- "DB_Data_F4_Btt_Down_Selected"
   Rectangle "Rectangle_3" at 25,1214 size 41x54
      VerticalMovement <- "Simu_Eleveytor"
      Visibility <- "Simu_Eleveytor"
   Button "Button_1" at 273,1218 size 25x24; TextOff '^'
      on Press: SetBit("DB_Data_F1_I_Button_Up")
      on Release: ResetBit("DB_Data_F1_I_Button_Up")
      Appearance <- "DB_Data_F1_Btt_Up_Selected"
   Button "Button_2" at 273,1106 size 25x24; TextOff '^'
      on Press: SetBit("DB_Data_F2_I_Button_Up")
      on Release: ResetBit("DB_Data_F2_I_Button_Up")
      Appearance <- "DB_Data_F2_Btt_Up_Selected"
   Button "Button_3" at 273,1082 size 25x24; TextOff 'v'
      on Press: SetBit("DB_Data_F2_I_Button_Down")
      on Release: ResetBit("DB_Data_F2_I_Button_Down")
      Appearance <- "DB_Data_F2_Btt_Down_Selected"
   Button "Button_4" at 273,986 size 25x24; TextOff '^'
      on Press: SetBit("DB_Data_F3_I_Button_Up")
      on Release: ResetBit("DB_Data_F3_I_Button_Up")
      Appearance <- "DB_Data_F3_Btt_Up_Selected"
   Button "Button_5" at 273,962 size 25x24; TextOff 'v'
      on Press: SetBit("DB_Data_F3_I_Button_Down")
      on Release: ResetBit("DB_Data_F3_I_Button_Down")
      Appearance <- "DB_Data_F3_Btt_Down_Selected"
   Button "Button_30" at 273,719 size 25x24; TextOff 'v'
      on Release: ResetBit("DB_Data_F5_I_Button_Down")
      on Press: SetBit("DB_Data_F5_I_Button_Down")
      Appearance <- "DB_Data_F5_Btt_Down_Selected"
   Button "Button_31" at 272,739 size 25x24; TextOff '^'
      on Release: ResetBit("DB_Data_F5_I_Button_Up")
      on Press: SetBit("DB_Data_F5_I_Button_Up")
      Appearance <- "DB_Data_F5_Btt_Up_Selected"
   Button "Button_29" at 272,869 size 25x24; TextOff '^'
      on Release: ResetBit("DB_Data_F4_I_Button_Up")
      on Press: SetBit("DB_Data_F4_I_Button_Up")
      Appearance <- "DB_Data_F4_Btt_Up_Selected"
   Button "Button_32" at 272,600 size 25x24; TextOff 'v'
      on Release: ResetBit("DB_Data_F6_I_Button_Down")
      on Press: SetBit("DB_Data_F6_I_Button_Down")
      Appearance <- "DB_Data_F6_Btt_Down_Selected"
   Button "Button_33" at 272,621 size 25x24; TextOff '^'
      on Release: ResetBit("DB_Data_F6_I_Button_Up")
      on Press: SetBit("DB_Data_F6_I_Button_Up")
      Appearance <- "DB_Data_F6_Btt_Up_Selected"
   Button "Button_36" at 275,360 size 25x24; TextOff 'v'
      on Release: ResetBit("DB_Data_F2_I_Button_Down")
      on Press: SetBit("DB_Data_F2_I_Button_Down")
      Appearance <- "DB_Data_F2_Btt_Down_Selected"
   Button "Button_37" at 275,264 size 25x24; TextOff '^'
      on Release: ResetBit("DB_Data_F3_I_Button_Up")
      on Press: SetBit("DB_Data_F3_I_Button_Up")
      Appearance <- "DB_Data_F3_Btt_Up_Selected"
   Button "Button_38" at 275,240 size 25x24; TextOff 'v'
      on Release: ResetBit("DB_Data_F3_I_Button_Down")
      on Press: SetBit("DB_Data_F3_I_Button_Down")
      Appearance <- "DB_Data_F3_Btt_Down_Selected"
   Button "Button_41" at 594,1209 size 25x24; TextOff 'v'
      on Release: ResetBit("DB_Data_F5_I_Button_Down")
      on Press: SetBit("DB_Data_F5_I_Button_Down")
      Appearance <- "DB_Data_F5_Btt_Down_Selected"
   Button "Button_45" at 275,497 size 25x24; TextOff '^'
      on Release: ResetBit("DB_Data_F7_I_Button_Up")
      on Press: SetBit("DB_Data_F7_I_Button_Up")
      Appearance <- "DB_Data_F7_Btt_Up_Selected"
   Button "Button_46" at 275,366 size 25x24; TextOff '^'
      on Release: ResetBit("DB_Data_F8_I_Button_Up")
      on Press: SetBit("DB_Data_F8_I_Button_Up")
      Appearance <- "DB_Data_F8_Btt_Up_Selected"
   Button "Button_47" at 275,342 size 25x24; TextOff 'v'
      on Release: ResetBit("DB_Data_F8_I_Button_Down")
      on Press: SetBit("DB_Data_F8_I_Button_Down")
      Appearance <- "DB_Data_F8_Btt_Down_Selected"
   Button "Button_48" at 275,264 size 25x24; TextOff '^'
      on Release: ResetBit("DB_Data_F9_I_Button_Up")
      on Press: SetBit("DB_Data_F9_I_Button_Up")
      Appearance <- "DB_Data_F9_Btt_Up_Selected"
   Button "Button_49" at 275,240 size 25x24; TextOff 'v'
      on Release: ResetBit("DB_Data_F9_I_Button_Down")
      on Press: SetBit("DB_Data_F9_I_Button_Down")
      Appearance <- "DB_Data_F3_Btt_Down_Selected"
   Button "Button_50" at 275,116 size 25x24; TextOff 'v'
      on Release: ResetBit("DB_Data_F10_I_Button_Down")
      on Press: SetBit("DB_Data_F10_I_Button_Down")
      Appearance <- "DB_Data_F10_Btt_Down_Selected"
   Rectangle "Rectangle_92" at 337,1217 size 41x54
      Visibility <- "Simu_Eleveytor"
      VerticalMovement <- "Simu_Eleveytor"
   Button "Button_51" at 275,139 size 25x24; TextOff '^'
      on Release: ResetBit("DB_Data_F10_I_Button_Up")
      on Press: SetBit("DB_Data_F10_I_Button_Up")
      Appearance <- "DB_Data_F10_Btt_Up_Selected"
   Button "Button_52" at 594,1185 size 25x24; TextOff 'v'
      on Release: ResetBit("DB_Data_F11_I_Button_Down")
      on Press: SetBit("DB_Data_F11_I_Button_Down")
      Appearance <- "DB_Data_F11_Btt_Down_Selected"
   Button "Button_53" at 593,1215 size 25x24; TextOff '^'
      on Release: ResetBit("DB_Data_F11_I_Button_Up")
      on Press: SetBit("DB_Data_F11_I_Button_Up")
      Appearance <- "DB_Data_F11_Btt_Up_Selected"
   Button "Button_54" at 591,1070 size 25x24; TextOff 'v'
      on Release: ResetBit("DB_Data_F12_I_Button_Down")
      on Press: SetBit("DB_Data_F12_I_Button_Down")
      Appearance <- "DB_Data_F12_Btt_Down_Selected"
   Button "Button_55" at 591,1095 size 25x24; TextOff '^'
      on Release: ResetBit("DB_Data_F12_I_Button_Up")
      on Press: SetBit("DB_Data_F12_I_Button_Up")
      Appearance <- "DB_Data_F12_Btt_Up_Selected"
   Button "Button_56" at 593,977 size 25x24; TextOff '^'
      on Release: ResetBit("DB_Data_F13_I_Button_Up")
      on Press: SetBit("DB_Data_F13_I_Button_Up")
      Appearance <- "DB_Data_F13_Btt_Up_Selected"
   Button "Button_57" at 593,858 size 25x24; TextOff '^'
      on Release: ResetBit("DB_Data_F14_I_Button_Up")
      on Press: SetBit("DB_Data_F14_I_Button_Up")
      Appearance <- "DB_Data_F14_Btt_Up_Selected"
   Button "Button_58" at 593,834 size 25x24; TextOff 'v'
      on Release: ResetBit("DB_Data_F14_I_Button_Down")
      on Press: SetBit("DB_Data_F14_I_Button_Down")
      Appearance <- "DB_Data_F14_Btt_Down_Selected"
   Button "Button_59" at 593,730 size 25x24; TextOff '^'
      on Release: ResetBit("DB_Data_F15_I_Button_Up")
      on Press: SetBit("DB_Data_F15_I_Button_Up")
      Appearance <- "DB_Data_F15_Btt_Up_Selected"
   Button "Button_60" at 593,706 size 25x24; TextOff 'v'
      on Release: ResetBit("DB_Data_F15_I_Button_Down")
      on Press: SetBit("DB_Data_F15_I_Button_Down")
      Appearance <- "DB_Data_F15_Btt_Down_Selected"
   Button "Button_61" at 592,607 size 25x24; TextOff 'v'
      on Release: ResetBit("DB_Data_F16_I_Button_Down")
      on Press: SetBit("DB_Data_F16_I_Button_Down")
      Appearance <- "DB_Data_F16_Btt_Down_Selected"
   Button "Button_62" at 592,631 size 25x24; TextOff '^'
      on Release: ResetBit("DB_Data_F16_I_Button_Up")
      on Press: SetBit("DB_Data_F16_I_Button_Up")
      Appearance <- "DB_Data_F16_Btt_Up_Selected"
   Button "Button_67" at 275,473 size 25x24; TextOff 'v'
      on Release: ResetBit("DB_Data_F7_I_Button_Down")
      on Press: SetBit("DB_Data_F7_I_Button_Down")
      Appearance <- "DB_Data_F7_Btt_Down_Selected"
   Button "Button_68" at 593,955 size 25x24; TextOff 'v'
      on Release: ResetBit("DB_Data_F13_I_Button_Down")
      on Press: SetBit("DB_Data_F13_I_Button_Down")
      Appearance <- "DB_Data_F13_Btt_Down_Selected"
   Button "Button_34" at 600,480 size 25x24; TextOff 'v'
      on Release: ResetBit("DB_Data_F17_I_Button_Down")
      on Press: SetBit("DB_Data_F17_I_Button_Down")
      Appearance <- "DB_Data_F17_Btt_Down_Selected"
   Button "Button_35" at 600,504 size 25x24; TextOff '^'
      on Release: ResetBit("DB_Data_F17_I_Button_Up")
      on Press: SetBit("DB_Data_F17_I_Button_Up")
      Appearance <- "DB_Data_F17_Btt_Up_Selected"
   Button "Button_39" at 593,345 size 25x24; TextOff 'v'
      on Release: ResetBit("DB_Data_F18_I_Button_Down")
      on Press: SetBit("DB_Data_F18_I_Button_Down")
      Appearance <- "DB_Data_F18_Btt_Down_Selected"
   Button "Button_40" at 593,369 size 25x24; TextOff '^'
      on Release: ResetBit("DB_Data_F18_I_Button_Up")
      on Press: SetBit("DB_Data_F18_I_Button_Up")
      Appearance <- "DB_Data_F18_Btt_Up_Selected"
   Button "Button_42" at 593,230 size 25x24; TextOff 'v'
      on Release: ResetBit("DB_Data_F19_I_Button_Down")
      on Press: SetBit("DB_Data_F19_I_Button_Down")
      Appearance <- "DB_Data_F19_Btt_Down_Selected"
   Button "Button_43" at 593,254 size 25x24; TextOff '^'
      on Release: ResetBit("DB_Data_F19_I_Button_Up")
      on Press: SetBit("DB_Data_F19_I_Button_Up")
      Appearance <- "DB_Data_F19_Btt_Up_Selected"
   Button "Button_44" at 593,115 size 25x24; TextOff 'v'
      on Release: ResetBit("DB_Data_F20_I_Button_Down")
      on Press: SetBit("DB_Data_F20_I_Button_Down")
      Appearance <- "DB_Data_F20_Btt_Down_Selected"
   Rectangle "Rectangle_97" at 411,687 size 78x102
      HorizontalMovement <- "Simu_Door_F15"
   Rectangle "Rectangle_98" at 488,687 size 78x102
      HorizontalMovement <- "Simu_Door_F15"
   Rectangle "Rectangle_99" at 411,567 size 78x102
      HorizontalMovement <- "Simu_Door_F16"
   Rectangle "Rectangle_100" at 488,567 size 78x102
      HorizontalMovement <- "Simu_Door_F16"
   Rectangle "Rectangle_113" at 409,443 size 78x102
      HorizontalMovement <- "Simu_Door_F17"
   Rectangle "Rectangle_114" at 486,443 size 78x102
      HorizontalMovement <- "Simu_Door_F17"
   Rectangle "Rectangle_118" at 411,318 size 78x102
      HorizontalMovement <- "Simu_Door_F18"
   Rectangle "Rectangle_119" at 488,318 size 78x102
      HorizontalMovement <- "Simu_Door_F18"
   Rectangle "Rectangle_2" at 411,203 size 78x102
      HorizontalMovement <- "Simu_Door_F19"
   Rectangle "Rectangle_21" at 488,203 size 78x102
      HorizontalMovement <- "Simu_Door_F19"
   Rectangle "Rectangle_37" at 411,88 size 78x102
      HorizontalMovement <- "Simu_Door_F20"
   Rectangle "Rectangle_38" at 488,88 size 78x102
      HorizontalMovement <- "Simu_Door_F20"
   Rectangle "Rectangle_95" at 411,807 size 78x102
      HorizontalMovement <- "Simu_Door_F14"
   Rectangle "Rectangle_96" at 488,807 size 78x102
      HorizontalMovement <- "Simu_Door_F14"
   Rectangle "Rectangle_94" at 486,923 size 78x102
      HorizontalMovement <- "Simu_Door_F13"
   Rectangle "Rectangle_93" at 412,924 size 78x102
      HorizontalMovement <- "Simu_Door_F13"
   Rectangle "Rectangle_4" at 91,1168 size 78x102
      HorizontalMovement <- "Simu_Door_F1"
   Rectangle "Rectangle_5" at 168,1168 size 78x102
      HorizontalMovement <- "Simu_Door_F1"
   Rectangle "Rectangle_6" at 91,1048 size 78x102
      HorizontalMovement <- "Simu_Door_F2"
   Rectangle "Rectangle_7" at 168,1048 size 78x102
      HorizontalMovement <- "Simu_Door_F2"
   Rectangle "Rectangle_8" at 91,928 size 78x102
      HorizontalMovement <- "Simu_Door_F3"
   Rectangle "Rectangle_9" at 168,928 size 78x102
      HorizontalMovement <- "Simu_Door_F3"
   Rectangle "Rectangle_10" at 91,808 size 78x102
      HorizontalMovement <- "Simu_Door_F4"
   Rectangle "Rectangle_11" at 168,808 size 78x102
      HorizontalMovement <- "Simu_Door_F4"
   Button "Button_6" at 708,45 size 57x26; TextOff 'F1'
      on Press: SetBit("DB_Data_Button_Inside_F1")
      on Release: ResetBit("DB_Data_Button_Inside_F1")
      Appearance <- "DB_Data_F1_Btt_Up_Selected"
   Button "Button_8" at 708,77 size 57x26; TextOff 'F2'
      on Press: SetBit("DB_Data_Button_Inside_F2")
      on Release: ResetBit("DB_Data_Button_Inside_F2")
      Appearance <- "Display_Inside_F2"
   Button "Button_9" at 708,109 size 57x26; TextOff 'F3'
      on Press: SetBit("DB_Data_Button_Inside_F3")
      on Release: ResetBit("DB_Data_Button_Inside_F3")
      Appearance <- "Display_Inside_F3"
   Button "Button_10" at 708,141 size 57x26; TextOff 'F4'
      on Press: SetBit("DB_Data_Button_Inside_F4")
      on Release: ResetBit("DB_Data_Button_Inside_F4")
      Appearance <- "Display_Inside_F4"
   Button "Button_11" at 855,80 size 57x26; TextOff 'MỞ'
      on Press: SetBit("DB_Data_Button_Inside_Open")
      on Release: ResetBit("DB_Data_Button_Inside_Open")
      Appearance <- "Q_Door_Open"
   Button "Button_12" at 855,45 size 57x26; TextOff 'ĐÓNG'
      on Press: SetBit("DB_Data_Button_Inside_Close")
      on Release: ResetBit("DB_Data_Button_Inside_Close")
      Appearance <- "Q_Door_Close"
   Switch "Switch_1" at 753,700 size 164x64; CaptionText 'MÔ PHỎNG'; TextOff 'OFF'; TextOn 'ON'
      ProcessValue <- "M_Simulation"
      on SwitchOn: SetBit("M_Simulation")
      on SwitchOff: ResetBit("M_Simulation")
   Rectangle "Rectangle_23" at 74,1254 size 15x12
      Appearance <- "DB_Data_F1_Sensor_Correct_Position"
   Rectangle "Rectangle_24" at 74,1133 size 15x12
      Appearance <- "DB_Data_F2_Sensor_Correct_Position"
   Rectangle "Rectangle_25" at 74,1012 size 15x12
      Appearance <- "DB_Data_F3_Sensor_Correct_Position"
   Rectangle "Rectangle_26" at 74,891 size 15x12
      Appearance <- "DB_Data_F4_Sensor_Correct_Position"
   Button "Button_13" at 708,177 size 57x26; TextOff 'F5'
      on Release: ResetBit("DB_Data_Button_Inside_F5")
      on Press: SetBit("DB_Data_Button_Inside_F5")
      Appearance <- "Display_Inside_F5"
   Button "Button_17" at 789,45 size 57x26; TextOff 'F11'
      on Release: ResetBit("DB_Data_Button_Inside_F11")
      on Press: SetBit("DB_Data_Button_Inside_F11")
      Appearance <- "Display_Inside_F11"
   Button "Button_18" at 789,77 size 57x26; TextOff 'F12'
      on Release: ResetBit("DB_Data_Button_Inside_F12")
      on Press: SetBit("DB_Data_Button_Inside_F12")
      Appearance <- "Display_Inside_F12"
   Button "Button_19" at 789,109 size 57x26; TextOff 'F13'
      on Release: ResetBit("DB_Data_Button_Inside_F13")
      on Press: SetBit("DB_Data_Button_Inside_F13")
      Appearance <- "Display_Inside_F13"
   Button "Button_20" at 789,141 size 57x26; TextOff 'F14'
      on Release: ResetBit("DB_Data_Button_Inside_F14")
      on Press: SetBit("DB_Data_Button_Inside_F14")
      Appearance <- "Display_Inside_F14"
   Button "Button_21" at 789,177 size 57x26; TextOff 'F15'
      on Release: ResetBit("DB_Data_Button_Inside_F15")
      on Press: SetBit("DB_Data_Button_Inside_F15")
      Appearance <- "Display_Inside_F15"
   Rectangle "Rectangle_27" at 91,687 size 78x102
      HorizontalMovement <- "Simu_Door_F5"
   Rectangle "Rectangle_28" at 168,687 size 78x102
      HorizontalMovement <- "Simu_Door_F5"
   Rectangle "Rectangle_31" at 76,783 size 15x12
      Appearance <- "DB_Data_F5_Sensor_Correct_Position"
   Rectangle "Rectangle_29" at 91,559 size 78x102
      HorizontalMovement <- "Simu_Door_F6"
   Rectangle "Rectangle_32" at 168,559 size 78x102
      HorizontalMovement <- "Simu_Door_F6"
   Rectangle "Rectangle_34" at 76,655 size 15x12
      Appearance <- "DB_Data_F6_Sensor_Correct_Position"
   Rectangle "Rectangle_50" at 76,528 size 15x12
      Appearance <- "DB_Data_F1_Sensor_Correct_Position"
   Rectangle "Rectangle_13" at 93,439 size 84x105
      HorizontalMovement <- "Simu_Door_F7"
   Rectangle "Rectangle_64" at 169,442 size 78x102
      HorizontalMovement <- "Simu_Door_F7"
   Rectangle "Rectangle_51" at 76,407 size 15x12
      Appearance <- "DB_Data_F2_Sensor_Correct_Position"
   Rectangle "Rectangle_52" at 76,286 size 15x12
      Appearance <- "DB_Data_F3_Sensor_Correct_Position"
   Rectangle "Rectangle_65" at 94,325 size 78x102
      HorizontalMovement <- "Simu_Door_F8"
   Rectangle "Rectangle_53" at 76,165 size 15x12
      Appearance <- "DB_Data_F4_Sensor_Correct_Position"
   Rectangle "Rectangle_66" at 171,325 size 78x102
      HorizontalMovement <- "Simu_Door_F8"
   Rectangle "Rectangle_67" at 92,205 size 78x102
      HorizontalMovement <- "Simu_Door_F9"
   Rectangle "Rectangle_68" at 169,205 size 78x102
      HorizontalMovement <- "Simu_Door_F9"
   Rectangle "Rectangle_69" at 91,85 size 78x102
      HorizontalMovement <- "Simu_Door_F10"
   Rectangle "Rectangle_70" at 169,86 size 78x102
      HorizontalMovement <- "Simu_Door_F10"
   Rectangle "Rectangle_79" at 76,528 size 15x12
      Appearance <- "DB_Data_F7_Sensor_Correct_Position"
   Rectangle "Rectangle_84" at 487,1168 size 78x102
      HorizontalMovement <- "Simu_Door_F11"
   Rectangle "Rectangle_83" at 410,1168 size 78x102
      HorizontalMovement <- "Simu_Door_F11"
   Rectangle "Rectangle_88" at 411,1045 size 78x102
      HorizontalMovement <- "Simu_Door_F12"
   Rectangle "Rectangle_89" at 488,1049 size 78x98
      HorizontalMovement <- "Simu_Door_F12"
   Rectangle "Rectangle_80" at 76,407 size 15x12
      Appearance <- "DB_Data_F8_Sensor_Correct_Position"
   Rectangle "Rectangle_81" at 76,286 size 15x12
      Appearance <- "DB_Data_F9_Sensor_Correct_Position"
   Rectangle "Rectangle_82" at 76,165 size 15x12
      Appearance <- "DB_Data_F10_Sensor_Correct_Position"
   Rectangle "Rectangle_86" at 392,1253 size 15x12
      Appearance <- "DB_Data_F11_Sensor_Correct_Position"
   Rectangle "Rectangle_91" at 393,1132 size 15x12
      Appearance <- "DB_Data_F12_Sensor_Correct_Position"
   Rectangle "Rectangle_110" at 394,892 size 15x12
      Appearance <- "DB_Data_F14_Sensor_Correct_Position"
   Rectangle "Rectangle_111" at 394,771 size 15x12
      Appearance <- "DB_Data_F15_Sensor_Correct_Position"
   Rectangle "Rectangle_112" at 394,650 size 15x12
      Appearance <- "DB_Data_F16_Sensor_Correct_Position"
   Rectangle "Rectangle_116" at 394,533 size 15x12
      Appearance <- "DB_Data_F17_Sensor_Correct_Position"
   Rectangle "Rectangle_121" at 393,396 size 15x12
      Appearance <- "DB_Data_F18_Sensor_Correct_Position"
   TextField "Text field_1" at 159,1211 size 15x22; Text '1'
   TextField "Text field_2" at 159,1092 size 15x22; Text '2'
   TextField "Text field_4" at 159,973 size 15x22; Text '3'
   TextField "Text field_5" at 159,854 size 15x22; Text '4'
   TextField "Text field_6" at 159,735 size 15x22; Text '5'
   TextField "Text field_7" at 159,616 size 15x22; Text '6'
   TextField "Text field_8" at 478,1102 size 29x22; Text '12'
   TextField "Text field_11" at 159,487 size 15x22; Text '7'
   TextField "Text field_13" at 158,367 size 15x22; Text '8'
   TextField "Text field_14" at 157,247 size 19x22; Text '9'
   TextField "Text field_15" at 156,127 size 29x22; Text '10'
   TextField "Text field_16" at 474,1201 size 29x22; Text '11'
   TextField "Text field_19" at 474,853 size 29x22; Text '14'
   TextField "Text field_20" at 469,733 size 29x22; Text '15'
   TextField "Text field_17" at 479,973 size 29x22; Text '13'
   TextField "Text field_21" at 468,612 size 29x22; Text '16'
   TextField "Text field_22" at 473,486 size 29x22; Text '17'
   TextField "Text field_23" at 473,359 size 29x22; Text '18'
   Rectangle "Rectangle_1" at 394,1005 size 15x12
      Appearance <- "DB_Data_F13_Sensor_Correct_Position"
   Rectangle "Rectangle_36" at 393,281 size 15x12
      Appearance <- "DB_Data_F19_Sensor_Correct_Position"
   TextField "Text field_9" at 473,244 size 29x22; Text '19'
   Rectangle "Rectangle_40" at 393,166 size 15x12
      Appearance <- "DB_Data_F20_Sensor_Correct_Position"
   TextField "Text field_10" at 473,129 size 29x22; Text '20'
   Button "Button_64" at 708,218 size 57x26; TextOff 'F6'
      on Release: ResetBit("DB_Data_Button_Inside_F6")
      on Press: SetBit("DB_Data_Button_Inside_F6")
      Appearance <- "Display_Inside_F6"
   Button "Button_65" at 708,259 size 57x26; TextOff 'F7'
      on Release: ResetBit("DB_Data_Button_Inside_F7")
      on Press: SetBit("DB_Data_Button_Inside_F7")
      Appearance <- "Display_Inside_F7"
   Button "Button_14" at 708,302 size 57x26; TextOff 'F8'
      on Release: ResetBit("DB_Data_Button_Inside_F8")
      on Press: SetBit("DB_Data_Button_Inside_F8")
      Appearance <- "Display_Inside_F8"
   Button "Button_15" at 707,342 size 57x26; TextOff 'F9'
      on Release: ResetBit("DB_Data_Button_Inside_F9")
      on Press: SetBit("DB_Data_Button_Inside_F9")
      Appearance <- "Display_Inside_F9"
   Button "Button_16" at 707,382 size 57x26; TextOff 'F10'
      on Release: ResetBit("DB_Data_Button_Inside_F10")
      on Press: SetBit("DB_Data_Button_Inside_F10")
      Appearance <- "Display_Inside_F10"
   Button "Button_22" at 789,218 size 57x26; TextOff 'F16'
      on Release: ResetBit("DB_Data_Button_Inside_F16")
      on Press: SetBit("DB_Data_Button_Inside_F16")
      Appearance <- "Display_Inside_F16"
   Button "Button_23" at 789,259 size 57x26; TextOff 'F17'
      on Release: ResetBit("DB_Data_Button_Inside_F17")
      on Press: SetBit("DB_Data_Button_Inside_F17")
      Appearance <- "Display_Inside_F17"
   Button "Button_24" at 789,300 size 57x26; TextOff 'F18'
      on Release: ResetBit("DB_Data_Button_Inside_F18")
      on Press: SetBit("DB_Data_Button_Inside_F18")
      Appearance <- "Display_Inside_F18"
   Button "Button_25" at 789,341 size 57x26; TextOff 'F19'
      on Release: ResetBit("DB_Data_Button_Inside_F19")
      on Press: SetBit("DB_Data_Button_Inside_F19")
      Appearance <- "Display_Inside_F19"
   Button "Button_26" at 789,382 size 57x26; TextOff 'F20'
      on Release: ResetBit("DB_Data_Button_Inside_F20")
      on Press: SetBit("DB_Data_Button_Inside_F20")
      Appearance <- "DB_Data_F20_Btt_Down_Selected"
*)